REGION Network 11: Trilgoten (4) - Reset Drive
   // Reset van Drive Trilgoten (Drive 2)
   RUNG wire#powerrail
      Contact( "Tag_9" )
      R_Coil( "Drive_2_Auto" )
   END_RUNG
   // the same network as SCL:
   IF "Tag_9" THEN "Drive_2_Auto" := FALSE; END_IF;
END_REGION

REGION Network 12: Aanvoerwals (1) - Set Timing as Drive 1
   RUNG wire#powerrail
      Contact( "PLCMemory".TimingSettingOvername )
      Coil( "Overname_Linked_Drive1" )
   END_RUNG
   // the same network as SCL:
   "Overname_Linked_Drive1" := "PLCMemory".TimingSettingOvername;
END_REGION

REGION Network 13: Aanvoerwals (2) - Run Drive (linked to drive 1)
   RUNG wire#powerrail
      Contact( "Overname_Linked_Drive1" )
      Contact( "Drive_1_Auto" )
      Coil( "Drive_4_Auto" )
   END_RUNG
   // the same network as SCL:
   "Drive_4_Auto" := "Overname_Linked_Drive1" AND "Drive_1_Auto";
END_REGION

REGION Network 14: Aanvoerwals (3) - Set speed Drive 4 (Linked to drive 1)
   RUNG wire#powerrail
      Contact( "PLCMemory".SpeedSettingsTakeover )
      Contact( "Drive 1 Speed 1" )
      Coil( "Drive_4_Speed1_Link" )
   END_RUNG
   // the same network as SCL:
   "Drive_4_Speed1_Link" := "PLCMemory".SpeedSettingsTakeover AND "Drive 1 Speed 1";
END_REGION

REGION Network 15: Aanvoerwals (4) - Set alternative Speed 1
   RUNG wire#powerrail
      I_Contact( "PLCMemory".SpeedSettingsTakeover )
      Contact( "PLCMemory".SpeedSettingOvername )
      I_Contact( "Drive_RefuseLinkingDrive1" )
      Coil( "Drive_4_Speed1_Unlink" )
   END_RUNG
   // the same network as SCL:
   "Drive_4_Speed1_Unlink" := NOT "PLCMemory".SpeedSettingsTakeover AND "PLCMemory".SpeedSettingOvername AND NOT "Drive_RefuseLinkingDrive1";
END_REGION

REGION Network 16: Aanvoerwals (5) - Set alternative Speed 0
   RUNG wire#powerrail
      I_Contact( "PLCMemory".SpeedSettingsTakeover )
      I_Contact( "PLCMemory".SpeedSettingOvername )
      Coil( "Drive_RefuseLinkingDrive1" )
   END_RUNG
   // the same network as SCL:
   "Drive_RefuseLinkingDrive1" := NOT "PLCMemory".SpeedSettingsTakeover AND NOT "PLCMemory".SpeedSettingOvername;
END_REGION

REGION Network 17: Set Position Enable
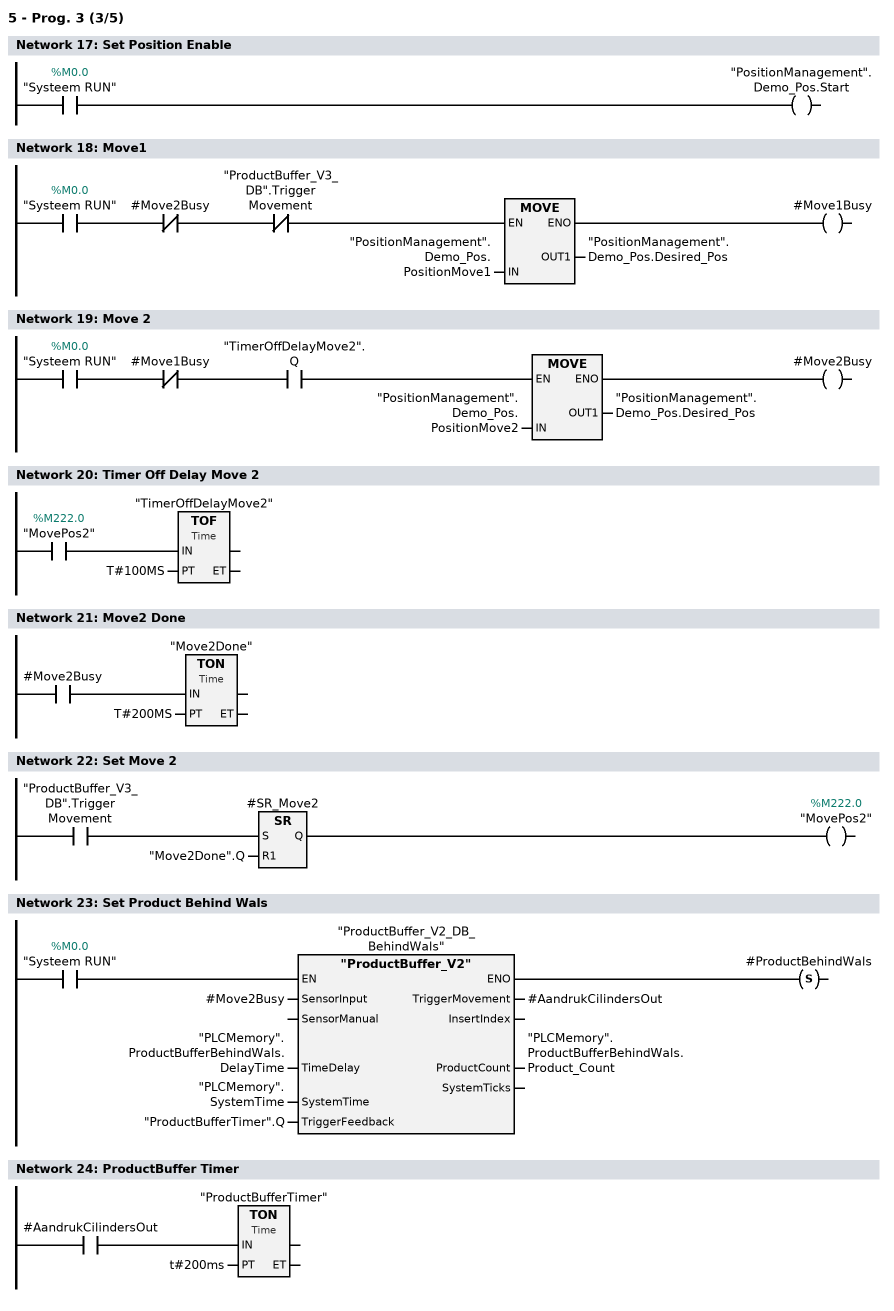
   RUNG wire#powerrail
      Contact( "Systeem RUN" )
      Coil( "PositionManagement".Demo_Pos.Start )
   END_RUNG
   // the same network as SCL:
   "PositionManagement".Demo_Pos.Start := "Systeem RUN";
END_REGION

REGION Network 18: Move1
   RUNG wire#powerrail
      Contact( "Systeem RUN" )
      I_Contact( #Move2Busy )
      I_Contact( "ProductBuffer_V3_DB".TriggerMovement )
      { S7_GenerateENO := "TRUE" } Move(in := "PositionManagement".Demo_Pos.PositionMove1, out1 => "PositionManagement".Demo_Pos.Desired_Pos)
      Coil( #Move1Busy )
   END_RUNG
   // the same network as SCL:
   // ENO of a box is taken as its EN; it also drops when the box reports an error
   #_w1 := "Systeem RUN" AND NOT #Move2Busy AND NOT "ProductBuffer_V3_DB".TriggerMovement;
   IF #_w1 THEN
       "PositionManagement".Demo_Pos.Desired_Pos := "PositionManagement".Demo_Pos.PositionMove1;
   END_IF;
   #Move1Busy := #_w1;
END_REGION

REGION Network 19: Move 2
   RUNG wire#powerrail
      Contact( "Systeem RUN" )
      I_Contact( #Move1Busy )
      Contact( "TimerOffDelayMove2".Q )
      { S7_GenerateENO := "TRUE" } Move(in := "PositionManagement".Demo_Pos.PositionMove2, out1 => "PositionManagement".Demo_Pos.Desired_Pos)
      Coil( #Move2Busy )
   END_RUNG
   // the same network as SCL:
   // ENO of a box is taken as its EN; it also drops when the box reports an error
   #_w1 := "Systeem RUN" AND NOT #Move1Busy AND "TimerOffDelayMove2".Q;
   IF #_w1 THEN
       "PositionManagement".Demo_Pos.Desired_Pos := "PositionManagement".Demo_Pos.PositionMove2;
   END_IF;
   #Move2Busy := #_w1;
END_REGION

REGION Network 20: Timer Off Delay Move 2
   RUNG wire#powerrail
      Contact( "MovePos2" )
      { S7_Templates := "time_type := Time" } "TimerOffDelayMove2".TOF(pt := T#100MS, et =>)
   END_RUNG
   // the same network as SCL:
   "TimerOffDelayMove2".TOF(IN := "MovePos2", PT := T#100MS);
END_REGION

REGION Network 21: Move2 Done
   RUNG wire#powerrail
      Contact( #Move2Busy )
      { S7_Templates := "time_type := Time" } "Move2Done".TON(pt := T#200MS, et =>)
   END_RUNG
   // the same network as SCL:
   "Move2Done".TON(IN := #Move2Busy, PT := T#200MS);
END_REGION

REGION Network 22: Set Move 2
   RUNG wire#powerrail
      Contact( "ProductBuffer_V3_DB".TriggerMovement )
      S_SR(operand := #SR_Move2, r1 := "Move2Done".Q)
      Coil( "MovePos2" )
   END_RUNG
   // the same network as SCL:
   IF "ProductBuffer_V3_DB".TriggerMovement THEN
       #SR_Move2 := TRUE;   // SR flip-flop
   END_IF;
   IF "Move2Done".Q THEN #SR_Move2 := FALSE; END_IF;
   "MovePos2" := #SR_Move2;
END_REGION

REGION Network 23: Set Product Behind Wals
   RUNG wire#powerrail
      Contact( "Systeem RUN" )
      "ProductBuffer_V2_DB_BehindWals"(SensorInput := #Move2Busy, SensorManual :=, TimeDelay := "PLCMemory".ProductBufferBehindWals.DelayTime, SystemTime := "PLCMemory".SystemTime, TriggerFeedback := "ProductBufferTimer".Q, TriggerMovement => #AandrukCilindersOut, InsertIndex =>, ProductCount => "PLCMemory".ProductBufferBehindWals.Product_Count, SystemTicks =>)
      S_Coil( #ProductBehindWals )
   END_RUNG
   // the same network as SCL:
   "ProductBuffer_V2_DB_BehindWals"(EN := "Systeem RUN",   // "ProductBuffer_V2"
                           SensorInput := #Move2Busy,
                           TimeDelay := "PLCMemory".ProductBufferBehindWals.DelayTime,
                           SystemTime := "PLCMemory".SystemTime,
                           TriggerFeedback := "ProductBufferTimer".Q,
                           TriggerMovement => #AandrukCilindersOut,
                           ProductCount => "PLCMemory".ProductBufferBehindWals.Product_Count,
                           ENO => #_w1);
   IF #_w1 THEN #ProductBehindWals := TRUE; END_IF;
END_REGION

REGION Network 24: ProductBuffer Timer
   RUNG wire#powerrail
      Contact( #AandrukCilindersOut )
      { S7_Templates := "time_type := Time" } "ProductBufferTimer".TON(pt := t#200ms, et =>)
   END_RUNG
   // the same network as SCL:
   "ProductBufferTimer".TON(IN := #AandrukCilindersOut, PT := t#200ms);
END_REGION

REGION Network 25: Aandrukken (3) - Outputs
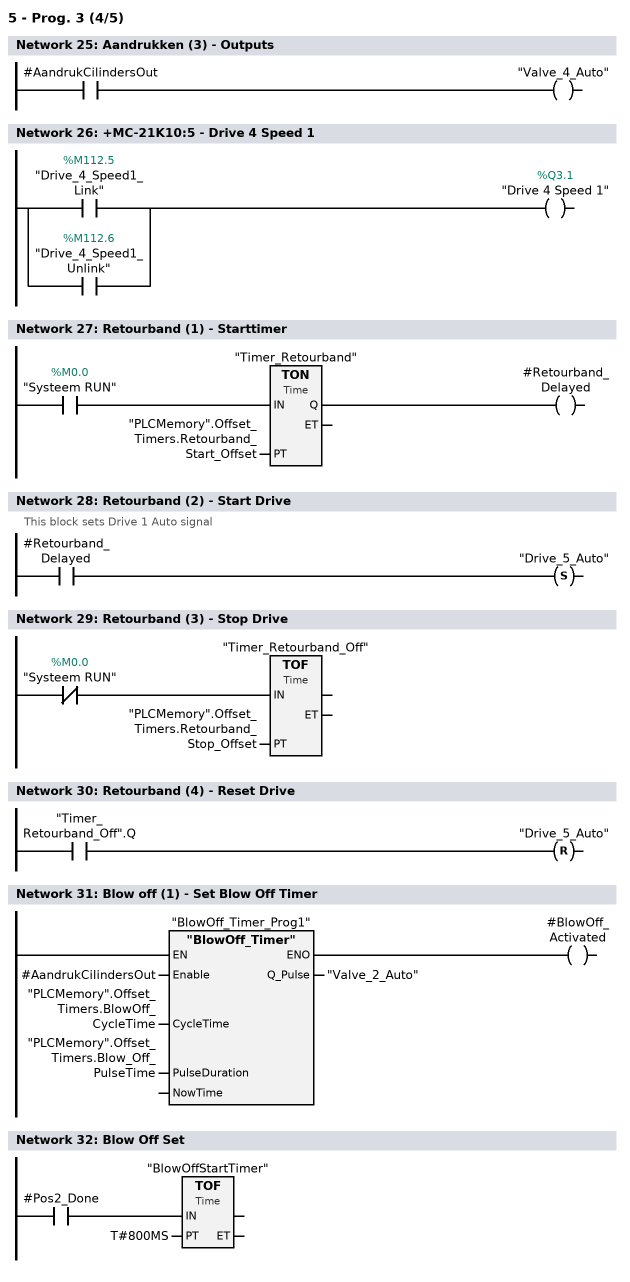
   RUNG wire#powerrail
      Contact( #AandrukCilindersOut )
      Coil( "Valve_4_Auto" )
   END_RUNG
   // the same network as SCL:
   "Valve_4_Auto" := #AandrukCilindersOut;
END_REGION

REGION Network 26: +MC-21K10:5 - Drive 4 Speed 1
   RUNG wire#powerrail
      Contact( "Drive_4_Speed1_Link" )
      wire#w1
      Coil( "Drive 4 Speed 1" )
   END_RUNG
   RUNG wire#powerrail
      Contact( "Drive_4_Speed1_Unlink" )
   END_RUNG wire#w1
   // the same network as SCL:
   "Drive 4 Speed 1" := "Drive_4_Speed1_Link" OR "Drive_4_Speed1_Unlink";
END_REGION

REGION Network 27: Retourband (1) - Starttimer
   RUNG wire#powerrail
      Contact( "Systeem RUN" )
      { S7_Templates := "time_type := Time" } "Timer_Retourband".TON(pt := "PLCMemory".Offset_Timers.Retourband_Start_Offset, et =>)
      Coil( #Retourband_Delayed )
   END_RUNG
   // the same network as SCL:
   "Timer_Retourband".TON(IN := "Systeem RUN", PT := "PLCMemory".Offset_Timers.Retourband_Start_Offset);
   #Retourband_Delayed := "Timer_Retourband".Q;
END_REGION

REGION Network 28: Retourband (2) - Start Drive
   // This block sets Drive 1 Auto signal
   RUNG wire#powerrail
      Contact( #Retourband_Delayed )
      S_Coil( "Drive_5_Auto" )
   END_RUNG
   // the same network as SCL:
   IF #Retourband_Delayed THEN "Drive_5_Auto" := TRUE; END_IF;
END_REGION

REGION Network 29: Retourband (3) - Stop Drive
   RUNG wire#powerrail
      I_Contact( "Systeem RUN" )
      { S7_Templates := "time_type := Time" } "Timer_Retourband_Off".TOF(pt := "PLCMemory".Offset_Timers.Retourband_Stop_Offset, et =>)
   END_RUNG
   // the same network as SCL:
   "Timer_Retourband_Off".TOF(IN := NOT "Systeem RUN", PT := "PLCMemory".Offset_Timers.Retourband_Stop_Offset);
END_REGION

REGION Network 30: Retourband (4) - Reset Drive
   RUNG wire#powerrail
      Contact( "Timer_Retourband_Off".Q )
      R_Coil( "Drive_5_Auto" )
   END_RUNG
   // the same network as SCL:
   IF "Timer_Retourband_Off".Q THEN "Drive_5_Auto" := FALSE; END_IF;
END_REGION

REGION Network 31: Blow off (1) - Set Blow Off Timer
   RUNG wire#powerrail
      "BlowOff_Timer_Prog1"(Enable := #AandrukCilindersOut, CycleTime := "PLCMemory".Offset_Timers.BlowOff_CycleTime, PulseDuration := "PLCMemory".Offset_Timers.Blow_Off_PulseTime, NowTime :=, Q_Pulse => "Valve_2_Auto")
      Coil( #BlowOff_Activated )
   END_RUNG
   // the same network as SCL:
   "BlowOff_Timer_Prog1"(Enable := #AandrukCilindersOut,   // "BlowOff_Timer"
                         CycleTime := "PLCMemory".Offset_Timers.BlowOff_CycleTime,
                         PulseDuration := "PLCMemory".Offset_Timers.Blow_Off_PulseTime,
                         Q_Pulse => "Valve_2_Auto",
                         ENO => #_w1);
   #BlowOff_Activated := #_w1;
END_REGION

REGION Network 32: Blow Off Set
   RUNG wire#powerrail
      Contact( #Pos2_Done )
      { S7_Templates := "time_type := Time" } "BlowOffStartTimer".TOF(pt := T#800MS, et =>)
   END_RUNG
   // the same network as SCL:
   "BlowOffStartTimer".TOF(IN := #Pos2_Done, PT := T#800MS);
END_REGION

REGION Network 33: BlowOffReset
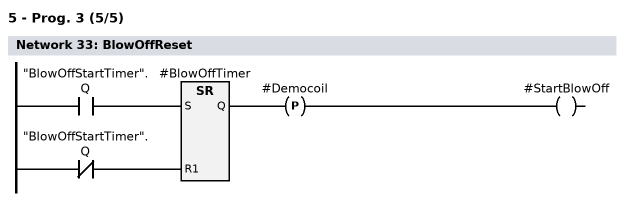
   RUNG wire#powerrail
      Contact( "BlowOffStartTimer".Q )
      S_SR(operand := #BlowOffTimer, r1 := wire#w1)
      P_Trig( #Democoil )
      Coil( #StartBlowOff )
   END_RUNG
   RUNG wire#powerrail
      I_Contact( "BlowOffStartTimer".Q )
   END_RUNG wire#w1
   // the same network as SCL:
   IF "BlowOffStartTimer".Q THEN
       #BlowOffTimer := TRUE;   // SR flip-flop
   END_IF;
   IF NOT "BlowOffStartTimer".Q THEN #BlowOffTimer := FALSE; END_IF;
   #_w1 := #BlowOffTimer AND NOT #Democoil;   // rising edge
   #Democoil := #BlowOffTimer;
   #StartBlowOff := #_w1;
END_REGION
END_FUNCTION

FUNCTION "1 - Outputs" : Void   // FC5, LAD
VERSION : 0.1
// This Function program is for operating the machine automatic and manual.
// stored: AutoNumber true, IsIECCheckEnabled false, UDAEnableTagReadback false
   VAR_TEMP
      Valve_2_Pulse : Bool;
      BlowOff_Activated : Bool;
      BlowOffManual : Bool;
      Pulse1 : Bool;
      Drive_1_ReferenceRun : Bool;
   END_VAR
   VAR_TEMP   // added for the SCL form of the ladder/FBD networks
      _w1 : Bool;
   END_VAR
BEGIN

REGION Network 1: Drive 1 - Control
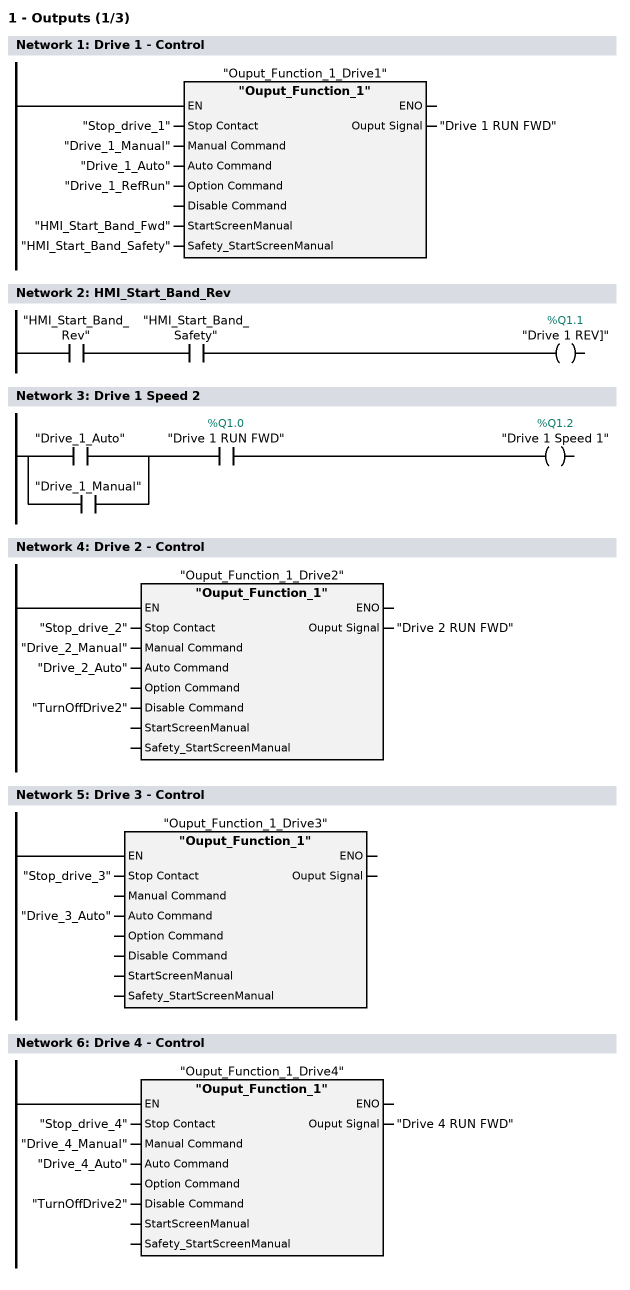
   RUNG wire#powerrail
      "Ouput_Function_1_Drive1"("Stop Contact" := "Stop_drive_1", "Manual Command" := "Drive_1_Manual", "Auto Command" := "Drive_1_Auto", "Option Command" := "Drive_1_RefRun", "Disable Command" :=, StartScreenManual := "HMI_Start_Band_Fwd", Safety_StartScreenManual := "HMI_Start_Band_Safety", "Ouput Signal" => "Drive 1 RUN FWD")
   END_RUNG
   // the same network as SCL:
   "Ouput_Function_1_Drive1"("Stop Contact" := "Stop_drive_1",   // "Ouput_Function_1"
                           "Manual Command" := "Drive_1_Manual",
                           "Auto Command" := "Drive_1_Auto",
                           "Option Command" := "Drive_1_RefRun",
                           StartScreenManual := "HMI_Start_Band_Fwd",
                           Safety_StartScreenManual := "HMI_Start_Band_Safety",
                           "Ouput Signal" => "Drive 1 RUN FWD");
END_REGION

REGION Network 2: HMI_Start_Band_Rev
   RUNG wire#powerrail
      Contact( "HMI_Start_Band_Rev" )
      Contact( "HMI_Start_Band_Safety" )
      Coil( "Drive 1 REV]" )
   END_RUNG
   // the same network as SCL:
   "Drive 1 REV]" := "HMI_Start_Band_Rev" AND "HMI_Start_Band_Safety";
END_REGION

REGION Network 3: Drive 1 Speed 2
   RUNG wire#powerrail
      Contact( "Drive_1_Auto" )
      wire#w1
      Contact( "Drive 1 RUN FWD" )
      Coil( "Drive 1 Speed 1" )
   END_RUNG
   RUNG wire#powerrail
      Contact( "Drive_1_Manual" )
   END_RUNG wire#w1
   // the same network as SCL:
   "Drive 1 Speed 1" := ("Drive_1_Auto" OR "Drive_1_Manual") AND "Drive 1 RUN FWD";
END_REGION

REGION Network 4: Drive 2 - Control
   RUNG wire#powerrail
      "Ouput_Function_1_Drive2"("Stop Contact" := "Stop_drive_2", "Manual Command" := "Drive_2_Manual", "Auto Command" := "Drive_2_Auto", "Option Command" :=, "Disable Command" := "TurnOffDrive2", StartScreenManual :=, Safety_StartScreenManual :=, "Ouput Signal" => "Drive 2 RUN FWD")
   END_RUNG
   // the same network as SCL:
   "Ouput_Function_1_Drive2"("Stop Contact" := "Stop_drive_2",   // "Ouput_Function_1"
                           "Manual Command" := "Drive_2_Manual",
                           "Auto Command" := "Drive_2_Auto",
                           "Disable Command" := "TurnOffDrive2",
                           "Ouput Signal" => "Drive 2 RUN FWD");
END_REGION

REGION Network 5: Drive 3 - Control
   RUNG wire#powerrail
      "Ouput_Function_1_Drive3"("Stop Contact" := "Stop_drive_3", "Manual Command" :=, "Auto Command" := "Drive_3_Auto", "Option Command" :=, "Disable Command" :=, StartScreenManual :=, Safety_StartScreenManual :=, "Ouput Signal" =>)
   END_RUNG
   // the same network as SCL:
   "Ouput_Function_1_Drive3"("Stop Contact" := "Stop_drive_3", "Auto Command" := "Drive_3_Auto");   // "Ouput_Function_1"
END_REGION

REGION Network 6: Drive 4 - Control
   RUNG wire#powerrail
      "Ouput_Function_1_Drive4"("Stop Contact" := "Stop_drive_4", "Manual Command" := "Drive_4_Manual", "Auto Command" := "Drive_4_Auto", "Option Command" :=, "Disable Command" := "TurnOffDrive2", StartScreenManual :=, Safety_StartScreenManual :=, "Ouput Signal" => "Drive 4 RUN FWD")
   END_RUNG
   // the same network as SCL:
   "Ouput_Function_1_Drive4"("Stop Contact" := "Stop_drive_4",   // "Ouput_Function_1"
                           "Manual Command" := "Drive_4_Manual",
                           "Auto Command" := "Drive_4_Auto",
                           "Disable Command" := "TurnOffDrive2",
                           "Ouput Signal" => "Drive 4 RUN FWD");
END_REGION

REGION Network 7: Drive 5 - Control
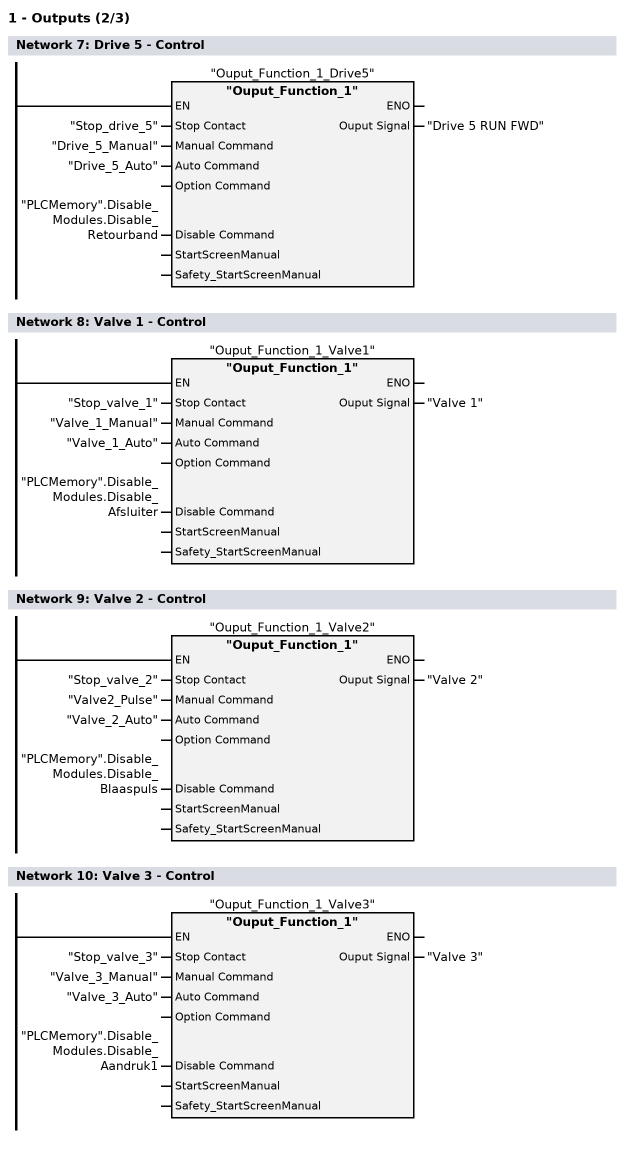
   RUNG wire#powerrail
      "Ouput_Function_1_Drive5"("Stop Contact" := "Stop_drive_5", "Manual Command" := "Drive_5_Manual", "Auto Command" := "Drive_5_Auto", "Option Command" :=, "Disable Command" := "PLCMemory".Disable_Modules.Disable_Retourband, StartScreenManual :=, Safety_StartScreenManual :=, "Ouput Signal" => "Drive 5 RUN FWD")
   END_RUNG
   // the same network as SCL:
   "Ouput_Function_1_Drive5"("Stop Contact" := "Stop_drive_5",   // "Ouput_Function_1"
                           "Manual Command" := "Drive_5_Manual",
                           "Auto Command" := "Drive_5_Auto",
                           "Disable Command" := "PLCMemory".Disable_Modules.Disable_Retourband,
                           "Ouput Signal" => "Drive 5 RUN FWD");
END_REGION

REGION Network 8: Valve 1 - Control
   RUNG wire#powerrail
      "Ouput_Function_1_Valve1"("Stop Contact" := "Stop_valve_1", "Manual Command" := "Valve_1_Manual", "Auto Command" := "Valve_1_Auto", "Option Command" :=, "Disable Command" := "PLCMemory".Disable_Modules.Disable_Afsluiter, StartScreenManual :=, Safety_StartScreenManual :=, "Ouput Signal" => "Valve 1")
   END_RUNG
   // the same network as SCL:
   "Ouput_Function_1_Valve1"("Stop Contact" := "Stop_valve_1",   // "Ouput_Function_1"
                           "Manual Command" := "Valve_1_Manual",
                           "Auto Command" := "Valve_1_Auto",
                           "Disable Command" := "PLCMemory".Disable_Modules.Disable_Afsluiter,
                           "Ouput Signal" => "Valve 1");
END_REGION

REGION Network 9: Valve 2 - Control
   RUNG wire#powerrail
      "Ouput_Function_1_Valve2"("Stop Contact" := "Stop_valve_2", "Manual Command" := "Valve2_Pulse", "Auto Command" := "Valve_2_Auto", "Option Command" :=, "Disable Command" := "PLCMemory".Disable_Modules.Disable_Blaaspuls, StartScreenManual :=, Safety_StartScreenManual :=, "Ouput Signal" => "Valve 2")
   END_RUNG
   // the same network as SCL:
   "Ouput_Function_1_Valve2"("Stop Contact" := "Stop_valve_2",   // "Ouput_Function_1"
                           "Manual Command" := "Valve2_Pulse",
                           "Auto Command" := "Valve_2_Auto",
                           "Disable Command" := "PLCMemory".Disable_Modules.Disable_Blaaspuls,
                           "Ouput Signal" => "Valve 2");
END_REGION

REGION Network 10: Valve 3 - Control
   RUNG wire#powerrail
      "Ouput_Function_1_Valve3"("Stop Contact" := "Stop_valve_3", "Manual Command" := "Valve_3_Manual", "Auto Command" := "Valve_3_Auto", "Option Command" :=, "Disable Command" := "PLCMemory".Disable_Modules.Disable_Aandruk1, StartScreenManual :=, Safety_StartScreenManual :=, "Ouput Signal" => "Valve 3")
   END_RUNG
   // the same network as SCL:
   "Ouput_Function_1_Valve3"("Stop Contact" := "Stop_valve_3",   // "Ouput_Function_1"
                           "Manual Command" := "Valve_3_Manual",
                           "Auto Command" := "Valve_3_Auto",
                           "Disable Command" := "PLCMemory".Disable_Modules.Disable_Aandruk1,
                           "Ouput Signal" => "Valve 3");
END_REGION

REGION Network 11: Valve 4 - Control
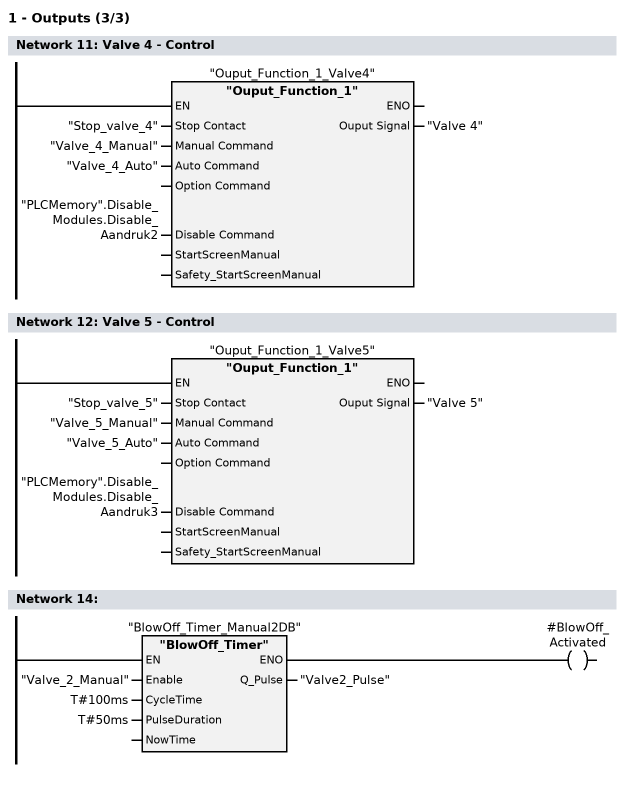
   RUNG wire#powerrail
      "Ouput_Function_1_Valve4"("Stop Contact" := "Stop_valve_4", "Manual Command" := "Valve_4_Manual", "Auto Command" := "Valve_4_Auto", "Option Command" :=, "Disable Command" := "PLCMemory".Disable_Modules.Disable_Aandruk2, StartScreenManual :=, Safety_StartScreenManual :=, "Ouput Signal" => "Valve 4")
   END_RUNG
   // the same network as SCL:
   "Ouput_Function_1_Valve4"("Stop Contact" := "Stop_valve_4",   // "Ouput_Function_1"
                           "Manual Command" := "Valve_4_Manual",
                           "Auto Command" := "Valve_4_Auto",
                           "Disable Command" := "PLCMemory".Disable_Modules.Disable_Aandruk2,
                           "Ouput Signal" => "Valve 4");
END_REGION

REGION Network 12: Valve 5 - Control
   RUNG wire#powerrail
      "Ouput_Function_1_Valve5"("Stop Contact" := "Stop_valve_5", "Manual Command" := "Valve_5_Manual", "Auto Command" := "Valve_5_Auto", "Option Command" :=, "Disable Command" := "PLCMemory".Disable_Modules.Disable_Aandruk3, StartScreenManual :=, Safety_StartScreenManual :=, "Ouput Signal" => "Valve 5")
   END_RUNG
   // the same network as SCL:
   "Ouput_Function_1_Valve5"("Stop Contact" := "Stop_valve_5",   // "Ouput_Function_1"
                           "Manual Command" := "Valve_5_Manual",
                           "Auto Command" := "Valve_5_Auto",
                           "Disable Command" := "PLCMemory".Disable_Modules.Disable_Aandruk3,
                           "Ouput Signal" => "Valve 5");
END_REGION

REGION Network 13: Blow Off Manual
END_REGION

REGION Network 14
   RUNG wire#powerrail
      "BlowOff_Timer_Manual2DB"(Enable := "Valve_2_Manual", CycleTime := T#100ms, PulseDuration := T#50ms, NowTime :=, Q_Pulse => "Valve2_Pulse")
      Coil( #BlowOff_Activated )
   END_RUNG
   // the same network as SCL:
   "BlowOff_Timer_Manual2DB"(Enable := "Valve_2_Manual",   // "BlowOff_Timer"
                           CycleTime := T#100ms,
                           PulseDuration := T#50ms,
                           Q_Pulse => "Valve2_Pulse",
                           ENO => #_w1);
   #BlowOff_Activated := #_w1;
END_REGION
END_FUNCTION

FUNCTION_BLOCK "Ouput_Function_1"   // FB8, FBD
TITLE = Ouput Controller Function Block
VERSION : 0.1
// stored: AutoNumber true, IsIECCheckEnabled false, UDAEnableTagReadback false
   VAR_INPUT
      "Stop Contact" : Bool;
      "Manual Command" : Bool;
      "Auto Command" : Bool;
      "Option Command" : Bool;
      "Disable Command" : Bool;
      StartScreenManual : Bool;
      Safety_StartScreenManual : Bool;
   END_VAR
   VAR_OUTPUT
      "Ouput Signal" : Bool;
   END_VAR
BEGIN

REGION Network 1: Ouput Controller
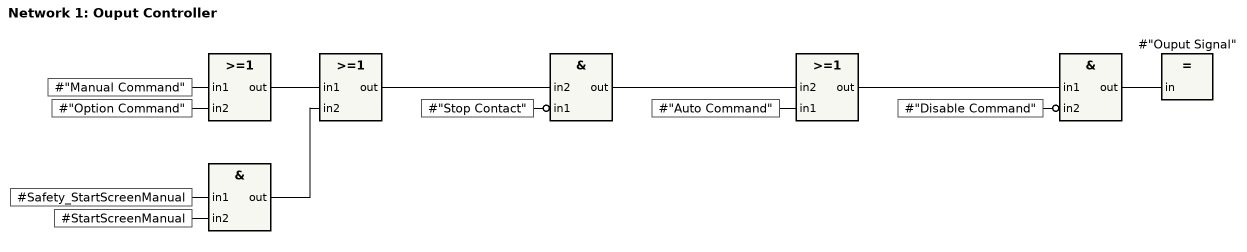
   #"Ouput Signal" := (((#"Manual Command" OR #"Option Command" OR (#Safety_StartScreenManual AND #StartScreenManual)) AND NOT #"Stop Contact") OR #"Auto Command") AND NOT #"Disable Command";
END_REGION
END_FUNCTION_BLOCK

FUNCTION "6 - Storingsmelding" : Void   // FC8, LAD
TITLE = Warnings
VERSION : 0.1
// This program block is for audible & visual warnings.
// stored: AutoNumber true, IsIECCheckEnabled false, UDAEnableTagReadback false
   VAR_TEMP
      "Wals Sensor Controlled" : Bool;
      "Infeed Sensor Controlled" : Bool;
      EnoughProductsOnInfeed : Bool;
      NotEnoughProductsOnInfeed : Bool;
      Warning_NotEnoughProducts : Bool;
      TurnOffDrives : Bool;
   END_VAR
   VAR CONSTANT
      "Sensor 2 (option)" : Bool := TRUE;
   END_VAR
   VAR_TEMP   // added for the SCL form of the ladder/FBD networks
      _w1 : Bool;
   END_VAR
BEGIN

REGION Network 1: +MC-21K6:5 - Bel Storing
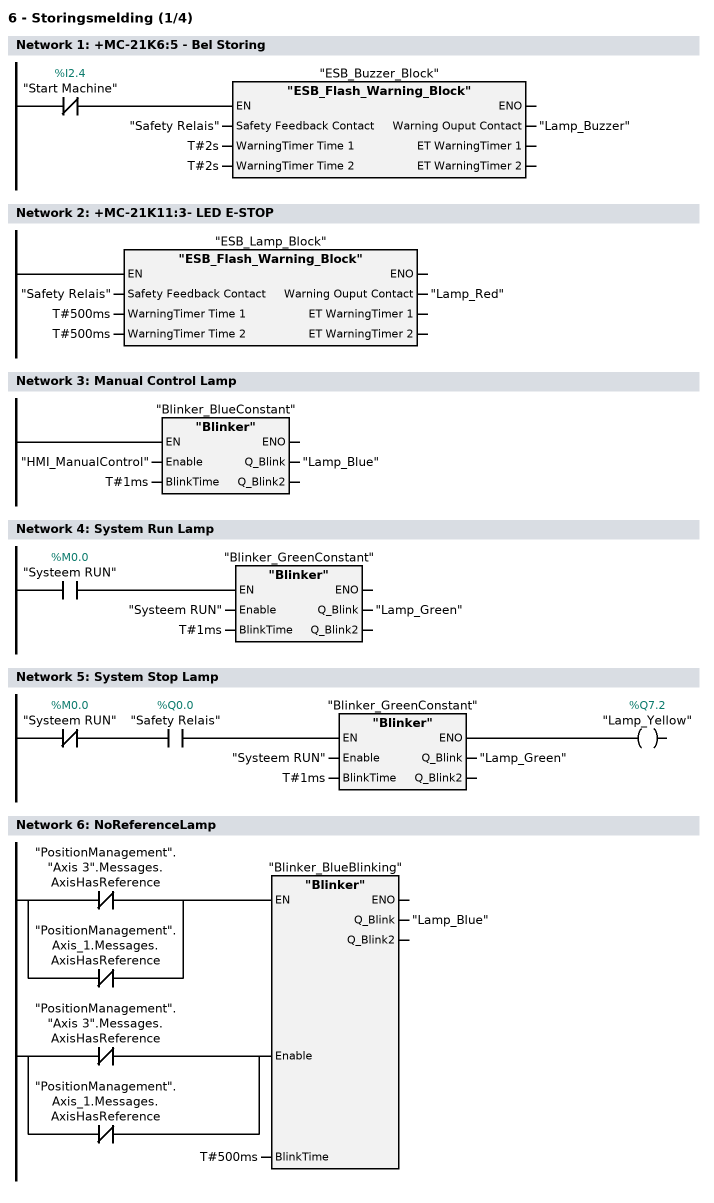
   RUNG wire#powerrail
      I_Contact( "Start Machine" )
      "ESB_Buzzer_Block"("Safety Feedback Contact" := "Safety Relais", "WarningTimer Time 1" := T#2s, "WarningTimer Time 2" := T#2s, "Warning Ouput Contact" => "Lamp_Buzzer", "ET WarningTimer 1" =>, "ET WarningTimer 2" =>)
   END_RUNG
   // the same network as SCL:
   IF NOT "Start Machine" THEN
       "ESB_Buzzer_Block"("Safety Feedback Contact" := "Safety Relais",   // "ESB_Flash_Warning_Block"
                          "WarningTimer Time 1" := T#2s,
                          "WarningTimer Time 2" := T#2s,
                          "Warning Ouput Contact" => "Lamp_Buzzer");
   END_IF;
END_REGION

REGION Network 2: +MC-21K11:3- LED E-STOP
   RUNG wire#powerrail
      "ESB_Lamp_Block"("Safety Feedback Contact" := "Safety Relais", "WarningTimer Time 1" := T#500ms, "WarningTimer Time 2" := T#500ms, "Warning Ouput Contact" => "Lamp_Red", "ET WarningTimer 1" =>, "ET WarningTimer 2" =>)
   END_RUNG
   // the same network as SCL:
   "ESB_Lamp_Block"("Safety Feedback Contact" := "Safety Relais",   // "ESB_Flash_Warning_Block"
                    "WarningTimer Time 1" := T#500ms,
                    "WarningTimer Time 2" := T#500ms,
                    "Warning Ouput Contact" => "Lamp_Red");
END_REGION

REGION Network 3: Manual Control Lamp
   RUNG wire#powerrail
      "Blinker_BlueConstant"(Enable := "HMI_ManualControl", BlinkTime := T#1ms, Q_Blink => "Lamp_Blue", Q_Blink2 =>)
   END_RUNG
   // the same network as SCL:
   "Blinker_BlueConstant"(Enable := "HMI_ManualControl", BlinkTime := T#1ms, Q_Blink => "Lamp_Blue");   // "Blinker"
END_REGION

REGION Network 4: System Run Lamp
   RUNG wire#powerrail
      Contact( "Systeem RUN" )
      "Blinker_GreenConstant"(Enable := "Systeem RUN", BlinkTime := T#1ms, Q_Blink => "Lamp_Green", Q_Blink2 =>)
   END_RUNG
   // the same network as SCL:
   IF "Systeem RUN" THEN
       "Blinker_GreenConstant"(Enable := "Systeem RUN", BlinkTime := T#1ms, Q_Blink => "Lamp_Green");   // "Blinker"
   END_IF;
END_REGION

REGION Network 5: System Stop Lamp
   RUNG wire#powerrail
      I_Contact( "Systeem RUN" )
      Contact( "Safety Relais" )
      "Blinker_GreenConstant"(Enable := "Systeem RUN", BlinkTime := T#1ms, Q_Blink => "Lamp_Green", Q_Blink2 =>)
      Coil( "Lamp_Yellow" )
   END_RUNG
   // the same network as SCL:
   "Blinker_GreenConstant"(EN := NOT "Systeem RUN" AND "Safety Relais",   // "Blinker"
                           Enable := "Systeem RUN",
                           BlinkTime := T#1ms,
                           Q_Blink => "Lamp_Green",
                           ENO => #_w1);
   "Lamp_Yellow" := #_w1;
END_REGION

REGION Network 6: NoReferenceLamp
   RUNG wire#powerrail
      I_Contact( "PositionManagement"."Axis 3".Messages.AxisHasReference )
      wire#w1
      "Blinker_BlueBlinking"(Enable := wire#w2, BlinkTime := T#500ms, Q_Blink => "Lamp_Blue", Q_Blink2 =>)
   END_RUNG
   RUNG wire#powerrail
      I_Contact( "PositionManagement".Axis_1.Messages.AxisHasReference )
   END_RUNG wire#w1
   RUNG wire#powerrail
      I_Contact( "PositionManagement"."Axis 3".Messages.AxisHasReference )
   END_RUNG wire#w2
   RUNG wire#powerrail
      I_Contact( "PositionManagement".Axis_1.Messages.AxisHasReference )
   END_RUNG wire#w2
   // the same network as SCL:
   IF NOT "PositionManagement"."Axis 3".Messages.AxisHasReference OR NOT "PositionManagement".Axis_1.Messages.AxisHasReference THEN
       "Blinker_BlueBlinking"(Enable := NOT "PositionManagement"."Axis 3".Messages.AxisHasReference OR NOT "PositionManagement".Axis_1.Messages.AxisHasReference,   // "Blinker"
                              BlinkTime := T#500ms,
                              Q_Blink => "Lamp_Blue");
   END_IF;
END_REGION

REGION Network 7: Fill Trechter Delay Function
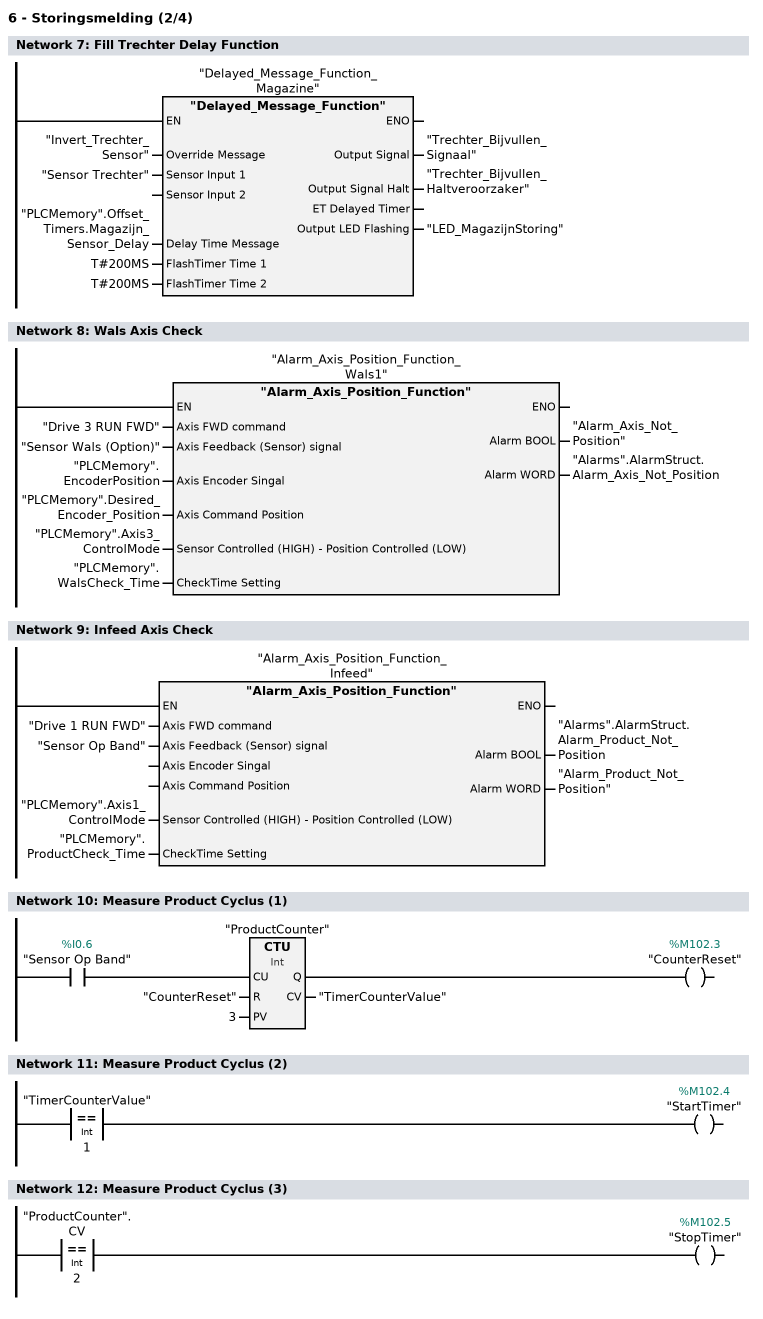
   RUNG wire#powerrail
      "Delayed_Message_Function_Magazine"("Override Message" := "Invert_Trechter_Sensor", "Sensor Input 1" := "Sensor Trechter", "Sensor Input 2" :=, "Delay Time Message" := "PLCMemory".Offset_Timers.Magazijn_Sensor_Delay, "FlashTimer Time 1" := T#200MS, "FlashTimer Time 2" := T#200MS, "Output Signal" => "Trechter_Bijvullen_Signaal", "Output Signal Halt" => "Trechter_Bijvullen_Haltveroorzaker", "ET Delayed Timer" =>, "Output LED Flashing" => "LED_MagazijnStoring")
   END_RUNG
   // the same network as SCL:
   "Delayed_Message_Function_Magazine"("Override Message" := "Invert_Trechter_Sensor",   // "Delayed_Message_Function"
                           "Sensor Input 1" := "Sensor Trechter",
                           "Delay Time Message" := "PLCMemory".Offset_Timers.Magazijn_Sensor_Delay,
                           "FlashTimer Time 1" := T#200MS,
                           "FlashTimer Time 2" := T#200MS,
                           "Output Signal" => "Trechter_Bijvullen_Signaal",
                           "Output Signal Halt" => "Trechter_Bijvullen_Haltveroorzaker",
                           "Output LED Flashing" => "LED_MagazijnStoring");
END_REGION

REGION Network 8: Wals Axis Check
   RUNG wire#powerrail
      "Alarm_Axis_Position_Function_Wals1"("Axis FWD command" := "Drive 3 RUN FWD", "Axis Feedback (Sensor) signal" := "Sensor Wals (Option)", "Axis Encoder Singal" := "PLCMemory".EncoderPosition, "Axis Command Position" := "PLCMemory".Desired_Encoder_Position, "Sensor Controlled (HIGH) - Position Controlled (LOW)" := "PLCMemory".Axis3_ControlMode, "CheckTime Setting" := "PLCMemory".WalsCheck_Time, "Alarm BOOL" => "Alarm_Axis_Not_Position", "Alarm WORD" => "Alarms".AlarmStruct.Alarm_Axis_Not_Position)
   END_RUNG
   // the same network as SCL:
   "Alarm_Axis_Position_Function_Wals1"("Axis FWD command" := "Drive 3 RUN FWD",   // "Alarm_Axis_Position_Function"
                           "Axis Feedback (Sensor) signal" := "Sensor Wals (Option)",
                           "Axis Encoder Singal" := "PLCMemory".EncoderPosition,
                           "Axis Command Position" := "PLCMemory".Desired_Encoder_Position,
                           "Sensor Controlled (HIGH) - Position Controlled (LOW)" := "PLCMemory".Axis3_ControlMode,
                           "CheckTime Setting" := "PLCMemory".WalsCheck_Time,
                           "Alarm BOOL" => "Alarm_Axis_Not_Position",
                           "Alarm WORD" => "Alarms".AlarmStruct.Alarm_Axis_Not_Position);
END_REGION

REGION Network 9: Infeed Axis Check
   RUNG wire#powerrail
      "Alarm_Axis_Position_Function_Infeed"("Axis FWD command" := "Drive 1 RUN FWD", "Axis Feedback (Sensor) signal" := "Sensor Op Band", "Axis Encoder Singal" :=, "Axis Command Position" :=, "Sensor Controlled (HIGH) - Position Controlled (LOW)" := "PLCMemory".Axis1_ControlMode, "CheckTime Setting" := "PLCMemory".ProductCheck_Time, "Alarm BOOL" => "Alarms".AlarmStruct.Alarm_Product_Not_Position, "Alarm WORD" => "Alarm_Product_Not_Position")
   END_RUNG
   // the same network as SCL:
   "Alarm_Axis_Position_Function_Infeed"("Axis FWD command" := "Drive 1 RUN FWD",   // "Alarm_Axis_Position_Function"
                           "Axis Feedback (Sensor) signal" := "Sensor Op Band",
                           "Sensor Controlled (HIGH) - Position Controlled (LOW)" := "PLCMemory".Axis1_ControlMode,
                           "CheckTime Setting" := "PLCMemory".ProductCheck_Time,
                           "Alarm BOOL" => "Alarms".AlarmStruct.Alarm_Product_Not_Position,
                           "Alarm WORD" => "Alarm_Product_Not_Position");
END_REGION

REGION Network 10: Measure Product Cyclus (1)
   RUNG wire#powerrail
      Contact( "Sensor Op Band" )
      { S7_Templates := "value_type := Int" } "ProductCounter".CTU(r := "CounterReset", pv := 3, cv => "TimerCounterValue")
      Coil( "CounterReset" )
   END_RUNG
   // the same network as SCL:
   "ProductCounter".CTU(CU := "Sensor Op Band", R := "CounterReset", PV := 3, CV => "TimerCounterValue");
   "CounterReset" := "ProductCounter".Q;
END_REGION

REGION Network 11: Measure Product Cyclus (2)
   RUNG wire#powerrail
      { S7_Templates := "SrcType := Int" } EQ_Contact(in1 := "TimerCounterValue", in2 := 1)
      Coil( "StartTimer" )
   END_RUNG
   // the same network as SCL:
   "StartTimer" := "TimerCounterValue" = 1;
END_REGION

REGION Network 12: Measure Product Cyclus (3)
   RUNG wire#powerrail
      { S7_Templates := "SrcType := Int" } EQ_Contact(in1 := "ProductCounter".CV, in2 := 2)
      Coil( "StopTimer" )
   END_RUNG
   // the same network as SCL:
   "StopTimer" := "ProductCounter".CV = 2;
END_REGION

REGION Network 13: Measure Product Cyclus (4)
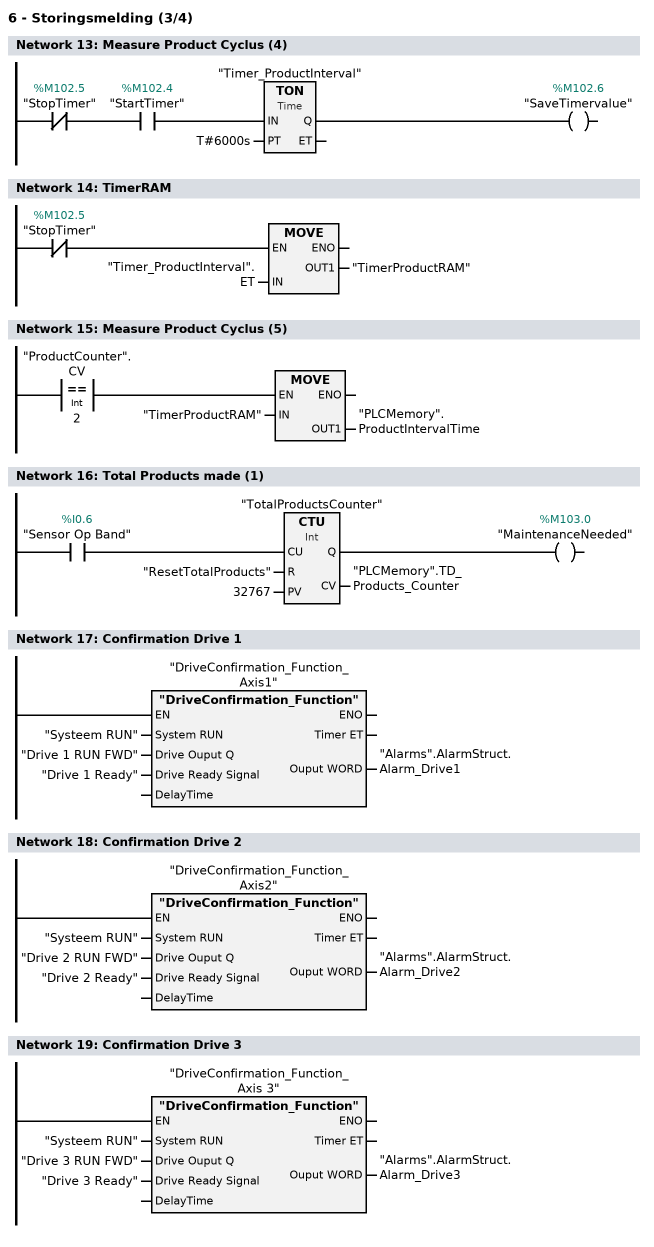
   RUNG wire#powerrail
      I_Contact( "StopTimer" )
      Contact( "StartTimer" )
      { S7_Templates := "time_type := Time" } "Timer_ProductInterval".TON(pt := T#6000s, et =>)
      Coil( "SaveTimervalue" )
   END_RUNG
   // the same network as SCL:
   "Timer_ProductInterval".TON(IN := NOT "StopTimer" AND "StartTimer", PT := T#6000s);
   "SaveTimervalue" := "Timer_ProductInterval".Q;
END_REGION

REGION Network 14: TimerRAM
   RUNG wire#powerrail
      I_Contact( "StopTimer" )
      { S7_GenerateENO := "TRUE" } Move(in := "Timer_ProductInterval".ET, out1 => "TimerProductRAM")
   END_RUNG
   // the same network as SCL:
   IF NOT "StopTimer" THEN "TimerProductRAM" := "Timer_ProductInterval".ET; END_IF;
END_REGION

REGION Network 15: Measure Product Cyclus (5)
   RUNG wire#powerrail
      { S7_Templates := "SrcType := Int" } EQ_Contact(in1 := "ProductCounter".CV, in2 := 2)
      { S7_GenerateENO := "TRUE" } Move(in := "TimerProductRAM", out1 => "PLCMemory".ProductIntervalTime)
   END_RUNG
   // the same network as SCL:
   IF "ProductCounter".CV = 2 THEN "PLCMemory".ProductIntervalTime := "TimerProductRAM"; END_IF;
END_REGION

REGION Network 16: Total Products made (1)
   RUNG wire#powerrail
      Contact( "Sensor Op Band" )
      { S7_Templates := "value_type := Int" } "TotalProductsCounter".CTU(r := "ResetTotalProducts", pv := 32767, cv => "PLCMemory".TD_Products_Counter)
      Coil( "MaintenanceNeeded" )
   END_RUNG
   // the same network as SCL:
   "TotalProductsCounter".CTU(CU := "Sensor Op Band",
                           R := "ResetTotalProducts",
                           PV := 32767,
                           CV => "PLCMemory".TD_Products_Counter);
   "MaintenanceNeeded" := "TotalProductsCounter".Q;
END_REGION

REGION Network 17: Confirmation Drive 1
   RUNG wire#powerrail
      "DriveConfirmation_Function_Axis1"("System RUN" := "Systeem RUN", "Drive Ouput Q" := "Drive 1 RUN FWD", "Drive Ready Signal" := "Drive 1 Ready", DelayTime :=, "Timer ET" =>, "Ouput WORD" => "Alarms".AlarmStruct.Alarm_Drive1)
   END_RUNG
   // the same network as SCL:
   "DriveConfirmation_Function_Axis1"("System RUN" := "Systeem RUN",   // "DriveConfirmation_Function"
                           "Drive Ouput Q" := "Drive 1 RUN FWD",
                           "Drive Ready Signal" := "Drive 1 Ready",
                           "Ouput WORD" => "Alarms".AlarmStruct.Alarm_Drive1);
END_REGION

REGION Network 18: Confirmation Drive 2
   RUNG wire#powerrail
      "DriveConfirmation_Function_Axis2"("System RUN" := "Systeem RUN", "Drive Ouput Q" := "Drive 2 RUN FWD", "Drive Ready Signal" := "Drive 2 Ready", DelayTime :=, "Timer ET" =>, "Ouput WORD" => "Alarms".AlarmStruct.Alarm_Drive2)
   END_RUNG
   // the same network as SCL:
   "DriveConfirmation_Function_Axis2"("System RUN" := "Systeem RUN",   // "DriveConfirmation_Function"
                           "Drive Ouput Q" := "Drive 2 RUN FWD",
                           "Drive Ready Signal" := "Drive 2 Ready",
                           "Ouput WORD" => "Alarms".AlarmStruct.Alarm_Drive2);
END_REGION

REGION Network 19: Confirmation Drive 3
   RUNG wire#powerrail
      "DriveConfirmation_Function_Axis 3"("System RUN" := "Systeem RUN", "Drive Ouput Q" := "Drive 3 RUN FWD", "Drive Ready Signal" := "Drive 3 Ready", DelayTime :=, "Timer ET" =>, "Ouput WORD" => "Alarms".AlarmStruct.Alarm_Drive3)
   END_RUNG
   // the same network as SCL:
   "DriveConfirmation_Function_Axis 3"("System RUN" := "Systeem RUN",   // "DriveConfirmation_Function"
                           "Drive Ouput Q" := "Drive 3 RUN FWD",
                           "Drive Ready Signal" := "Drive 3 Ready",
                           "Ouput WORD" => "Alarms".AlarmStruct.Alarm_Drive3);
END_REGION

REGION Network 20: Confimation Drive 4
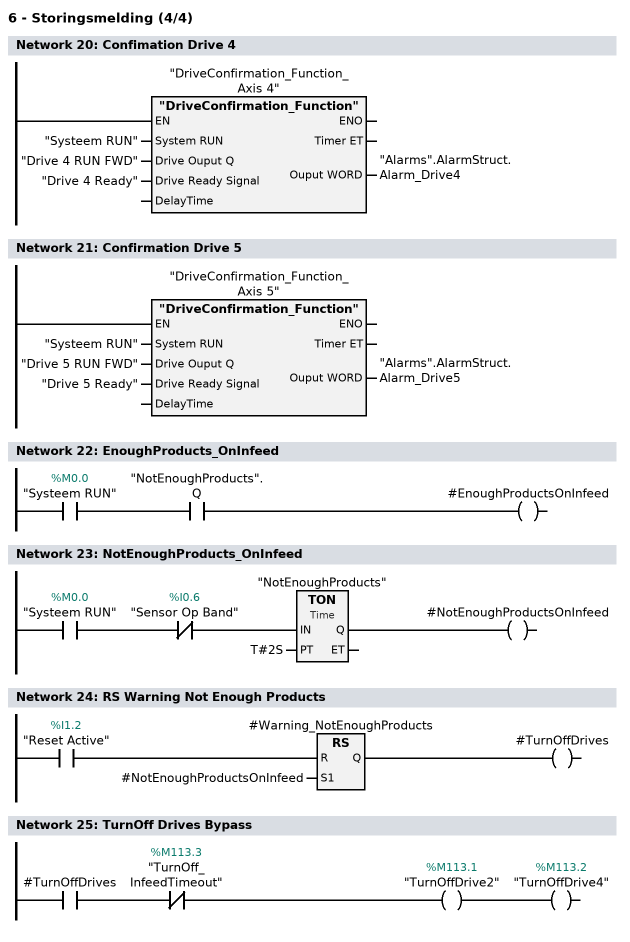
   RUNG wire#powerrail
      "DriveConfirmation_Function_Axis 4"("System RUN" := "Systeem RUN", "Drive Ouput Q" := "Drive 4 RUN FWD", "Drive Ready Signal" := "Drive 4 Ready", DelayTime :=, "Timer ET" =>, "Ouput WORD" => "Alarms".AlarmStruct.Alarm_Drive4)
   END_RUNG
   // the same network as SCL:
   "DriveConfirmation_Function_Axis 4"("System RUN" := "Systeem RUN",   // "DriveConfirmation_Function"
                           "Drive Ouput Q" := "Drive 4 RUN FWD",
                           "Drive Ready Signal" := "Drive 4 Ready",
                           "Ouput WORD" => "Alarms".AlarmStruct.Alarm_Drive4);
END_REGION

REGION Network 21: Confirmation Drive 5
   RUNG wire#powerrail
      "DriveConfirmation_Function_Axis 5"("System RUN" := "Systeem RUN", "Drive Ouput Q" := "Drive 5 RUN FWD", "Drive Ready Signal" := "Drive 5 Ready", DelayTime :=, "Timer ET" =>, "Ouput WORD" => "Alarms".AlarmStruct.Alarm_Drive5)
   END_RUNG
   // the same network as SCL:
   "DriveConfirmation_Function_Axis 5"("System RUN" := "Systeem RUN",   // "DriveConfirmation_Function"
                           "Drive Ouput Q" := "Drive 5 RUN FWD",
                           "Drive Ready Signal" := "Drive 5 Ready",
                           "Ouput WORD" => "Alarms".AlarmStruct.Alarm_Drive5);
END_REGION

REGION Network 22: EnoughProducts_OnInfeed
   RUNG wire#powerrail
      Contact( "Systeem RUN" )
      Contact( "NotEnoughProducts".Q )
      Coil( #EnoughProductsOnInfeed )
   END_RUNG
   // the same network as SCL:
   #EnoughProductsOnInfeed := "Systeem RUN" AND "NotEnoughProducts".Q;
END_REGION

REGION Network 23: NotEnoughProducts_OnInfeed
   RUNG wire#powerrail
      Contact( "Systeem RUN" )
      I_Contact( "Sensor Op Band" )
      { S7_Templates := "time_type := Time" } "NotEnoughProducts".TON(pt := T#2S, et =>)
      Coil( #NotEnoughProductsOnInfeed )
   END_RUNG
   // the same network as SCL:
   "NotEnoughProducts".TON(IN := "Systeem RUN" AND NOT "Sensor Op Band", PT := T#2S);
   #NotEnoughProductsOnInfeed := "NotEnoughProducts".Q;
END_REGION

REGION Network 24: RS Warning Not Enough Products
   RUNG wire#powerrail
      Contact( "Reset Active" )
      S_RS(operand := #Warning_NotEnoughProducts, s1 := #NotEnoughProductsOnInfeed)
      Coil( #TurnOffDrives )
   END_RUNG
   // the same network as SCL:
   IF "Reset Active" THEN
       #Warning_NotEnoughProducts := FALSE;   // RS flip-flop
   END_IF;
   IF #NotEnoughProductsOnInfeed THEN #Warning_NotEnoughProducts := TRUE; END_IF;
   #TurnOffDrives := #Warning_NotEnoughProducts;
END_REGION

REGION Network 25: TurnOff Drives Bypass
   RUNG wire#powerrail
      Contact( #TurnOffDrives )
      I_Contact( "TurnOff_InfeedTimeout" )
      Coil( "TurnOffDrive2" )
      Coil( "TurnOffDrive4" )
   END_RUNG
   // the same network as SCL:
   "TurnOffDrive2" := #TurnOffDrives AND NOT "TurnOff_InfeedTimeout";
   "TurnOffDrive4" := "TurnOffDrive2";
END_REGION
END_FUNCTION

FUNCTION_BLOCK "ESB_Flash_Warning_Block"   // FB1, FBD
VERSION : 0.1
// stored: AutoNumber true, IsIECCheckEnabled false, UDAEnableTagReadback false
   VAR_INPUT
      "Safety Feedback Contact" : Bool;
      "WarningTimer Time 1" : Time := T#150ms;
      "WarningTimer Time 2" : Time := T#150ms;
   END_VAR
   VAR_OUTPUT
      "Warning Ouput Contact" : Bool;
      "ET WarningTimer 1" : Time;
      "ET WarningTimer 2" : Time;
   END_VAR
   VAR_TEMP
      SafetyTakeoverContact : Bool;
   END_VAR
   VAR_TEMP   // added for the SCL form of the ladder/FBD networks
      _w1 : Bool;
   END_VAR
BEGIN

REGION Network 1: Flash Warning
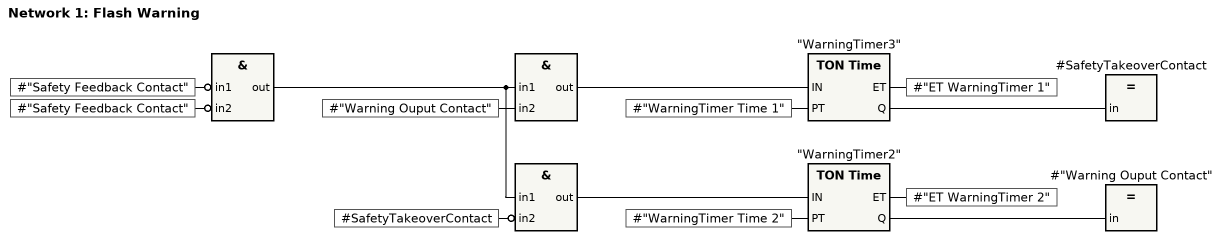
   #_w1 := NOT #"Safety Feedback Contact" AND NOT #"Safety Feedback Contact";
   "WarningTimer3".TON(IN := #_w1 AND #"Warning Ouput Contact",
                       PT := #"WarningTimer Time 1",
                       ET => #"ET WarningTimer 1");
   #SafetyTakeoverContact := "WarningTimer3".Q;
   "WarningTimer2".TON(IN := #_w1 AND NOT #SafetyTakeoverContact,
                       PT := #"WarningTimer Time 2",
                       ET => #"ET WarningTimer 2");
   #"Warning Ouput Contact" := "WarningTimer2".Q;
END_REGION
END_FUNCTION_BLOCK

FUNCTION_BLOCK "Delayed_Message_Function"   // FB2, FBD
TITLE = Delayed Message Function
VERSION : 0.1
// Functionblock For Delaying Message Function for example for filling an magazine or waiting for an signal. It is possible to adjust Time with the Dleay Time Message Input. The FlashTimer Time 1 & 2 ar for adjusting the flashing time of the ouput LED.
// stored: AutoNumber true, IsIECCheckEnabled false, UDAEnableTagReadback false
   VAR_INPUT
      "Override Message" : Bool;
      "Sensor Input 1" : Bool;
      "Sensor Input 2" : Bool := true;
      "Delay Time Message" : Time := T#1S_500MS;
      "FlashTimer Time 1" : Time := T#200ms;
      "FlashTimer Time 2" : Time := T#200ms;
   END_VAR
   VAR_OUTPUT
      "Output Signal" : Bool;
      "Output Signal Halt" : Bool;
      "ET Delayed Timer" : Time;
      "Output LED Flashing" : Bool;
   END_VAR
   VAR_TEMP
      "Internal Delayed Signal" : Bool;
   END_VAR
   VAR_TEMP   // added for the SCL form of the ladder/FBD networks
      _w1 : Bool;
   END_VAR
BEGIN

REGION Network 1: Delayed Signal to Outputs
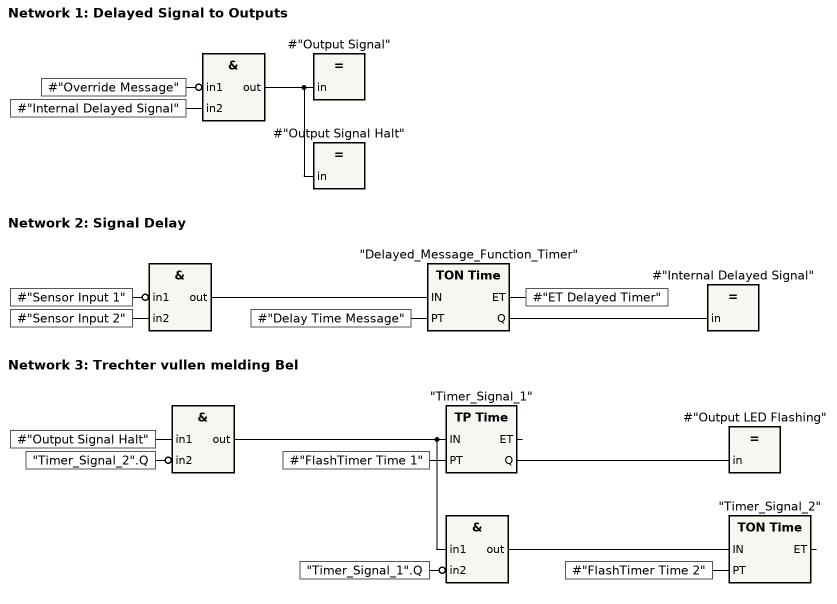
   #"Output Signal" := NOT #"Override Message" AND #"Internal Delayed Signal";
   #"Output Signal Halt" := #"Output Signal";
END_REGION

REGION Network 2: Signal Delay
   "Delayed_Message_Function_Timer".TON(IN := NOT #"Sensor Input 1" AND #"Sensor Input 2",
                           PT := #"Delay Time Message",
                           ET => #"ET Delayed Timer");
   #"Internal Delayed Signal" := "Delayed_Message_Function_Timer".Q;
END_REGION

REGION Network 3: Trechter vullen melding Bel
   #_w1 := #"Output Signal Halt" AND NOT "Timer_Signal_2".Q;
   "Timer_Signal_1".TP(IN := #_w1, PT := #"FlashTimer Time 1");
   #"Output LED Flashing" := "Timer_Signal_1".Q;
   "Timer_Signal_2".TON(IN := #_w1 AND NOT "Timer_Signal_1".Q, PT := #"FlashTimer Time 2");
END_REGION
END_FUNCTION_BLOCK

FUNCTION_BLOCK "Alarm_Axis_Position_Function"   // FB3, FBD
TITLE = Alarm Axis not in Position
VERSION : 0.1
// stored: AutoNumber true, IsIECCheckEnabled false, UDAEnableTagReadback false
   VAR_INPUT
      "Axis FWD command" : Bool;
      "Axis Feedback (Sensor) signal" : Bool;
      "Axis Encoder Singal" : Real;
      "Axis Command Position" : Real;
      "Sensor Controlled (HIGH) - Position Controlled (LOW)" : Bool;
      "CheckTime Setting" : Time := T#5S;
   END_VAR
   VAR_OUTPUT
      "Alarm BOOL" : Bool;
      "Alarm WORD" : Bool;
   END_VAR
   VAR_TEMP
      "Axis Feedback Internal" : Bool;
      "Axis Encoder On Position" : Bool;
      "Axis Sensor On Position" : Bool;
      "Axis Measuring Mode" : Bool;
   END_VAR
BEGIN

REGION Network 1: When axis is spinning start timer
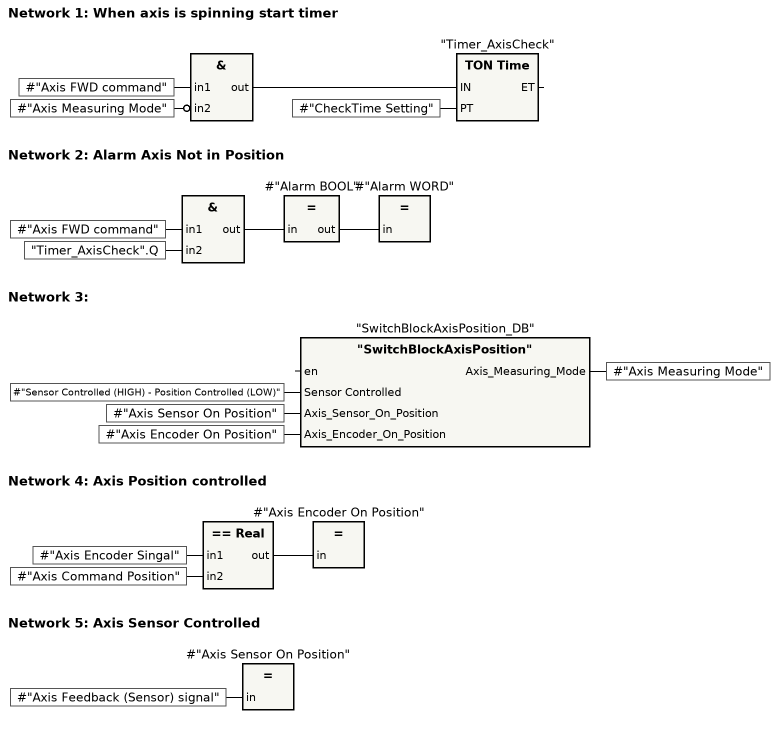
   "Timer_AxisCheck".TON(IN := #"Axis FWD command" AND NOT #"Axis Measuring Mode", PT := #"CheckTime Setting");
END_REGION

REGION Network 2: Alarm Axis Not in Position
   #"Alarm BOOL" := #"Axis FWD command" AND "Timer_AxisCheck".Q;
   #"Alarm WORD" := #"Alarm BOOL";
END_REGION

REGION Network 3
   "SwitchBlockAxisPosition_DB"("Sensor Controlled" := #"Sensor Controlled (HIGH) - Position Controlled (LOW)",   // "SwitchBlockAxisPosition"
                           Axis_Sensor_On_Position := #"Axis Sensor On Position",
                           Axis_Encoder_On_Position := #"Axis Encoder On Position",
                           Axis_Measuring_Mode => #"Axis Measuring Mode");
END_REGION

REGION Network 4: Axis Position controlled
   #"Axis Encoder On Position" := #"Axis Encoder Singal" = #"Axis Command Position";
END_REGION

REGION Network 5: Axis Sensor Controlled
   #"Axis Sensor On Position" := #"Axis Feedback (Sensor) signal";
END_REGION
END_FUNCTION_BLOCK

FUNCTION_BLOCK "SwitchBlockAxisPosition"
{ S7_Optimized_Access := 'FALSE' }
VERSION : 0.1
   VAR_INPUT 
      "Sensor Controlled" : Bool;
      Axis_Sensor_On_Position : Bool;
      Axis_Encoder_On_Position : Bool;
   END_VAR

   VAR_OUTPUT 
      Axis_Measuring_Mode : Bool;
   END_VAR


BEGIN
	IF #"Sensor Controlled" THEN
	    #Axis_Measuring_Mode := #Axis_Sensor_On_Position;
	ELSE
	    #Axis_Measuring_Mode := #Axis_Encoder_On_Position;
	END_IF;
	
END_FUNCTION_BLOCK

FUNCTION_BLOCK "DriveConfirmation_Function"   // FB5, FBD
TITLE = Drive Confirmation Function Block
VERSION : 0.1
// stored: AutoNumber true, IsIECCheckEnabled false, UDAEnableTagReadback false
   VAR_INPUT
      "System RUN" : Bool;
      "Drive Ouput Q" : Bool;
      "Drive Ready Signal" : Bool;
      DelayTime : Time := T#1s;
   END_VAR
   VAR_OUTPUT
      "Timer ET" : Time;
      "Ouput WORD" : Bool;
   END_VAR
BEGIN

REGION Network 1: Confirmation Drive
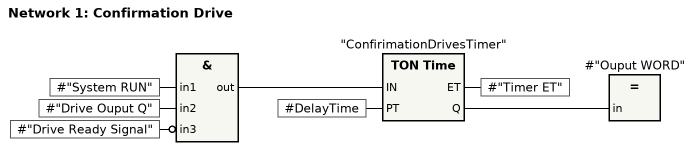
   "ConfirimationDrivesTimer".TON(IN := #"System RUN" AND #"Drive Ouput Q" AND NOT #"Drive Ready Signal",
                           PT := #DelayTime,
                           ET => #"Timer ET");
   #"Ouput WORD" := "ConfirimationDrivesTimer".Q;
END_REGION
END_FUNCTION_BLOCK

FUNCTION "9 - OVERIG" : Void   // FC6, LAD
TITLE = Other - Testing
VERSION : 0.1
// stored: AutoNumber true, IsIECCheckEnabled false, UDAEnableTagReadback false
   VAR_TEMP
      Encoder : Int;
      Gate : Bool;
      GATESTP : Bool;
      OTERRA : Bool;
      Direct : Bool;
      Prepar : Bool;
      CMPV1 : Bool;
      CMPV2 : Bool;
      RESSYNC : Bool;
      RESZERO : Bool;
      OTERR : Bool;
   END_VAR
BEGIN

REGION Network 1: SAFETY - OVERRIDE
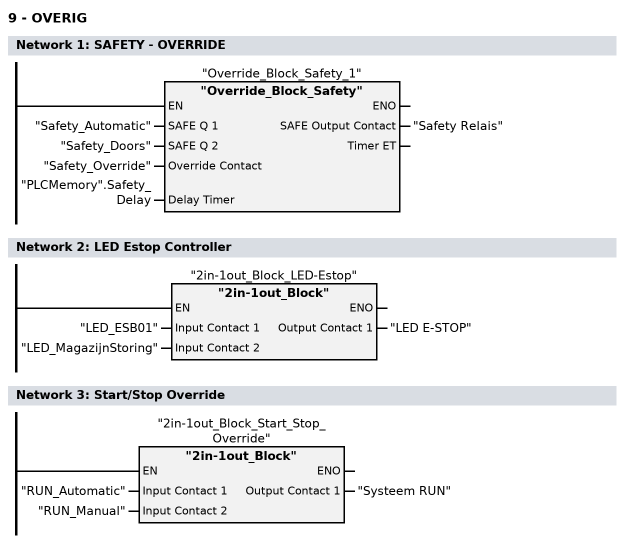
   RUNG wire#powerrail
      "Override_Block_Safety_1"("SAFE Q 1" := "Safety_Automatic", "SAFE Q 2" := "Safety_Doors", "Override Contact" := "Safety_Override", "Delay Timer" := "PLCMemory".Safety_Delay, "SAFE Output Contact" => "Safety Relais", "Timer ET" =>)
   END_RUNG
   // the same network as SCL:
   "Override_Block_Safety_1"("SAFE Q 1" := "Safety_Automatic",   // "Override_Block_Safety"
                           "SAFE Q 2" := "Safety_Doors",
                           "Override Contact" := "Safety_Override",
                           "Delay Timer" := "PLCMemory".Safety_Delay,
                           "SAFE Output Contact" => "Safety Relais");
END_REGION

REGION Network 2: LED Estop Controller
   RUNG wire#powerrail
      "2in-1out_Block_LED-Estop"("Input Contact 1" := "LED_ESB01", "Input Contact 2" := "LED_MagazijnStoring", "Output Contact 1" => "LED E-STOP")
   END_RUNG
   // the same network as SCL:
   "2in-1out_Block_LED-Estop"("Input Contact 1" := "LED_ESB01",   // "2in-1out_Block"
                           "Input Contact 2" := "LED_MagazijnStoring",
                           "Output Contact 1" => "LED E-STOP");
END_REGION

REGION Network 3: Start/Stop Override
   RUNG wire#powerrail
      "2in-1out_Block_Start_Stop_Override"("Input Contact 1" := "RUN_Automatic", "Input Contact 2" := "RUN_Manual", "Output Contact 1" => "Systeem RUN")
   END_RUNG
   // the same network as SCL:
   "2in-1out_Block_Start_Stop_Override"("Input Contact 1" := "RUN_Automatic",   // "2in-1out_Block"
                           "Input Contact 2" := "RUN_Manual",
                           "Output Contact 1" => "Systeem RUN");
END_REGION
END_FUNCTION

FUNCTION_BLOCK "Override_Block_Safety"   // FB7, FBD
TITLE = Override Block Safety.
VERSION : 0.1
// stored: AutoNumber true, IsIECCheckEnabled false, UDAEnableTagReadback false
   VAR_INPUT
      "SAFE Q 1" : Bool;
      "SAFE Q 2" : Bool;
      "Override Contact" : Bool;
      "Delay Timer" : Time;
   END_VAR
   VAR_OUTPUT
      "SAFE Output Contact" : Bool;
      "Timer ET" : Time;
   END_VAR
BEGIN

REGION Network 1: SAFETY - OVERRIDE
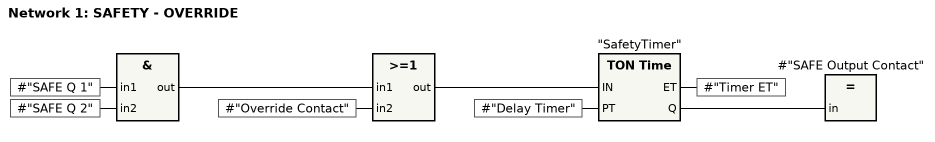
   "SafetyTimer".TON(IN := (#"SAFE Q 1" AND #"SAFE Q 2") OR #"Override Contact",
                     PT := #"Delay Timer",
                     ET => #"Timer ET");
   #"SAFE Output Contact" := "SafetyTimer".Q;
END_REGION
END_FUNCTION_BLOCK

FUNCTION_BLOCK "2in-1out_Block"   // FB6, FBD
VERSION : 0.1
// stored: AutoNumber true, IsIECCheckEnabled true, UDAEnableTagReadback false
   VAR_INPUT
      "Input Contact 1" : Bool;
      "Input Contact 2" : Bool;
   END_VAR
   VAR_OUTPUT
      "Output Contact 1" : Bool;
   END_VAR
BEGIN

REGION Network 1: Network Default
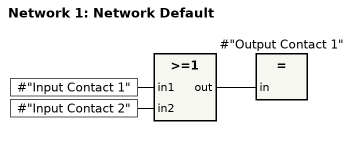
   #"Output Contact 1" := #"Input Contact 1" OR #"Input Contact 2";
END_REGION
END_FUNCTION_BLOCK

FUNCTION_BLOCK "ResetOuputs_Function"   // FB9, LAD
TITLE = Reset Ouput Functions With Commands
VERSION : 0.1
// stored: AutoNumber true, IsIECCheckEnabled false, UDAEnableTagReadback false
   VAR_INPUT
      StopCommand_NC : Bool;
      StopCommand_NO : Bool;
   END_VAR
   VAR_OUTPUT
      Output_1 : Bool;
      Output_2 : Bool;
      Output_3 : Bool;
      Output_4 : Bool;
      Output_5 : Bool;
      Output_6 : Bool;
      Output_7 : Bool;
      Output_8 : Bool;
      Output_9 : Bool;
      Output_10 : Bool;
   END_VAR
BEGIN

REGION Network 1: NW1
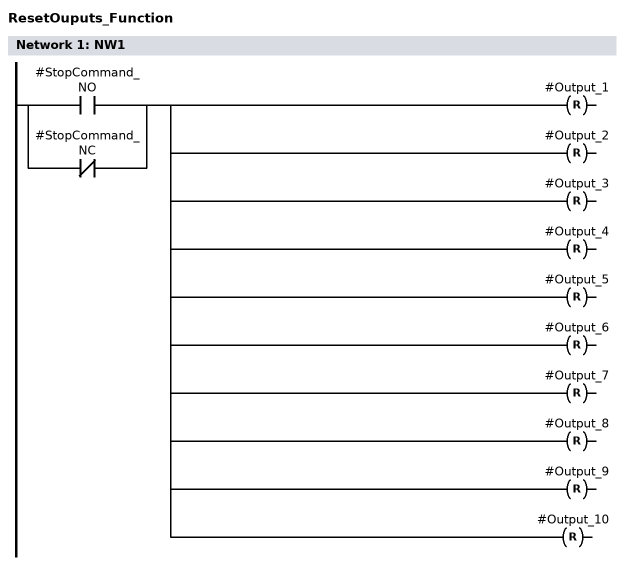
   RUNG wire#powerrail
      Contact( #StopCommand_NO )
      wire#w1
      R_Coil( #Output_1 )
   END_RUNG
   RUNG wire#powerrail
      I_Contact( #StopCommand_NC )
   END_RUNG wire#w1
   RUNG wire#w1
      R_Coil( #Output_2 )
   END_RUNG
   RUNG wire#w1
      R_Coil( #Output_3 )
   END_RUNG
   RUNG wire#w1
      R_Coil( #Output_4 )
   END_RUNG
   RUNG wire#w1
      R_Coil( #Output_5 )
   END_RUNG
   RUNG wire#w1
      R_Coil( #Output_6 )
   END_RUNG
   RUNG wire#w1
      R_Coil( #Output_7 )
   END_RUNG
   RUNG wire#w1
      R_Coil( #Output_8 )
   END_RUNG
   RUNG wire#w1
      R_Coil( #Output_9 )
   END_RUNG
   RUNG wire#w1
      R_Coil( #Output_10 )
   END_RUNG
   // the same network as SCL:
   IF #StopCommand_NO OR NOT #StopCommand_NC THEN
       #Output_1 := FALSE;
       #Output_2 := FALSE;
       #Output_3 := FALSE;
       #Output_4 := FALSE;
       #Output_5 := FALSE;
       #Output_6 := FALSE;
       #Output_7 := FALSE;
       #Output_8 := FALSE;
       #Output_9 := FALSE;
       #Output_10 := FALSE;
   END_IF;
END_REGION
END_FUNCTION_BLOCK

FUNCTION "SCL_Block" : Void
{ S7_Optimized_Access := 'FALSE' }
VERSION : 0.1

BEGIN
	// Reset de Word variabelen aan het begin van elke cyclus
	"Alarms".AlarmsWord := 0;
	"Alarms".HMI_Alarm_Drive1 := 0;
	"Alarms".HMI_Alarm_Drive2 := 0;
	"Alarms".HMI_Alarm_Drive3 := 0;
	"Alarms".HMI_Alarm_Drive4 := 0;
	"Alarms".HMI_Alarm_Drive5 := 0;
	
	// Controleer de alarmen en zet de respectievelijke bits aan
	IF "Alarms".AlarmStruct.Alarm_Product_Not_Position THEN
	    "Alarms".AlarmsWord := "Alarms".AlarmsWord OR WORD#1; // Zet bit 0 aan
	END_IF;
	
	IF "Alarms".AlarmStruct.Alarm_Axis_Not_Position THEN
	    "Alarms".AlarmsWord := "Alarms".AlarmsWord OR WORD#2; // Zet bit 1 aan
	END_IF;
	
	IF "Alarms".AlarmStruct.Alarm_Drive1 THEN
	    "Alarms".HMI_Alarm_Drive1 := "Alarms".HMI_Alarm_Drive1 OR WORD#1; // Zet bit 2 aan
	END_IF;
	
	IF "Alarms".AlarmStruct.Alarm_Drive2 THEN
	    "Alarms".HMI_Alarm_Drive2 := "Alarms".HMI_Alarm_Drive2 OR WORD#1; // Zet bit 3 aan
	END_IF;
	
	IF "Alarms".AlarmStruct.Alarm_Drive3 THEN
	    "Alarms".HMI_Alarm_Drive3 := "Alarms".HMI_Alarm_Drive3 OR WORD#1; // Zet bit 4 aan
	END_IF;
	
	IF "Alarms".AlarmStruct.Alarm_Drive4 THEN
	    "Alarms".HMI_Alarm_Drive4 := "Alarms".HMI_Alarm_Drive4 OR WORD#1; // Zet bit 5 aan
	END_IF;
	
	IF "Alarms".AlarmStruct.Alarm_Drive5 THEN
	    "Alarms".HMI_Alarm_Drive5 := "Alarms".HMI_Alarm_Drive5 OR WORD#1; // Zet bit 6 aan
	END_IF;
	
	
	// Position Program Axis 3 (Wals)
	
	// Configureer de timer om elke 0,5 seconde af te lopen
	"Timer_0_5s".TON(IN := TRUE,
	PT := "PLCMemory"."Encoder PulsOffset");
	
	// Controleer of de timer is afgelopen
	IF "Timer_0_5s".Q THEN
	    // Verhoog of verlaag de positie afhankelijk van de aandrijfsignalen
	    IF "Drive 3 RUN FWD" THEN
	        "PLCMemory".EncoderPosition := "PLCMemory".EncoderPosition + "PLCMemory".StepSize; // Verhoog met de stepgrootte
	    ELSIF "Drive 3 REV" THEN
	        "PLCMemory".EncoderPosition := "PLCMemory".EncoderPosition - "PLCMemory".StepSize; // Verlaag met de stepgrootte
	    END_IF;
	    
	    // Wrapping van de positie bij overschrijden van 360 graden of onder 0 graden
	    IF "PLCMemory".EncoderPosition >= 360.0 THEN
	        "PLCMemory".EncoderPosition := 0.0;  // Wrapping naar 0 als de positie 360 overschrijdt
	    ELSIF "PLCMemory".EncoderPosition < 0.0 THEN
	        "PLCMemory".EncoderPosition := 360.0; // Wrapping naar 360 als de positie onder 0 gaat
	    END_IF;
	    
	    // Reset de timer
	    "Timer_0_5s".TON (IN := FALSE,
	                      PT := "PLCMemory"."Encoder PulsOffset"); // Reset de timer zodat deze opnieuw kan starten
	END_IF;
	
	// Homing logica
	IF "Sensor Wals (Option)" THEN
	    "PLCMemory".EncoderPosition := 0.0;  // Reset de positie naar 0 als de sensor wordt geactiveerd
	END_IF;
	
	
	
	//Drive Servo Control Here:
	/// Desired Position Axis 3
	
	// Controleer of de HMI-knop is ingedrukt en er een gewenste positie is ingesteld
	//IF "HMI_Des_Pos_Axis3" THEN
	    //"GoButtonPressed" := TRUE; // HMI-knop is ingedrukt, start beweging
	//END_IF;
	
	// Beveiliging voor de Desired_Encoder_Position: Zorg dat de waarde tussen 0 en 360 blijft
	//IF "PLCMemory".Desired_Encoder_Position > 360.0 THEN
	  //  "PLCMemory".Desired_Encoder_Position := 360.0;  // Zet naar 360 als de waarde boven 360 ligt
	//ELSIF "PLCMemory".Desired_Encoder_Position < 0.0 THEN
	    //"PLCMemory".Desired_Encoder_Position := 0.0;  // Zet naar 0 als de waarde onder 0 ligt
	//END_IF;
	
	// Wrapping van de gewenste positie: Als de gewenste positie 360 is, zet deze dan op 0
	//IF "PLCMemory".Desired_Encoder_Position = 360.0 THEN
	   // "PLCMemory".Desired_Encoder_Position := 0.0;  // Wrapping naar 0 als de gewenste positie 360 is
	//END_IF;
	
	// Voer beweging uit totdat de gewenste positie is bereikt
	//IF "GoButtonPressed" THEN
	    // Bepaal de bewegingsrichting en start de beweging
	  //  IF "PLCMemory".EncoderPosition < "PLCMemory".Desired_Encoder_Position - "PLCMemory".Tolerance THEN
	        // Beweeg vooruit met StepSize als snelheid
	      //  "PLCMemory".EncoderPosition := "PLCMemory".EncoderPosition + "PLCMemory".StepSize;
	     //   "Drive_3_Manual" := TRUE;   // Activeer vooruitbeweging
	      //  "Drive 3 REV" := FALSE;     // Zorg dat achteruitbeweging uit is
	        
	  //  ELSIF "PLCMemory".EncoderPosition > "PLCMemory".Desired_Encoder_Position + "PLCMemory".Tolerance THEN
	        // Beweeg achteruit met StepSize als snelheid
	     //   "PLCMemory".EncoderPosition := "PLCMemory".EncoderPosition - "PLCMemory".StepSize;
	    //    "Drive_3_Manual" := FALSE;  // Zorg dat vooruitbeweging uit is
	    //    "Drive 3 REV" := TRUE;      // Activeer achteruitbeweging
	        
	   // ELSE
	        // Stop de beweging zodra de positie binnen de tolerantie komt
	      //  "Drive_3_Manual" := FALSE;    // Zet vooruitbeweging uit
	     //   "Drive 3 REV" := FALSE;       // Zet achteruitbeweging uit
	     //   "GoButtonPressed" := FALSE;   // Zet de Go-knop uit om verdere beweging te stoppen
	   // END_IF;
	//END_IF;
	
	
	
	
	
END_FUNCTION

FUNCTION "7 - Clean" : Void   // FC4, LAD
TITLE = Cleaning Program
VERSION : 0.1
// stored: AutoNumber true, IsIECCheckEnabled false, UDAEnableTagReadback false
   VAR_TEMP
      BlowOff_Active : Bool;
   END_VAR
   VAR_TEMP   // added for the SCL form of the ladder/FBD networks
      _w1 : Bool;
   END_VAR
BEGIN

REGION Network 1: Button Pressed Show Message
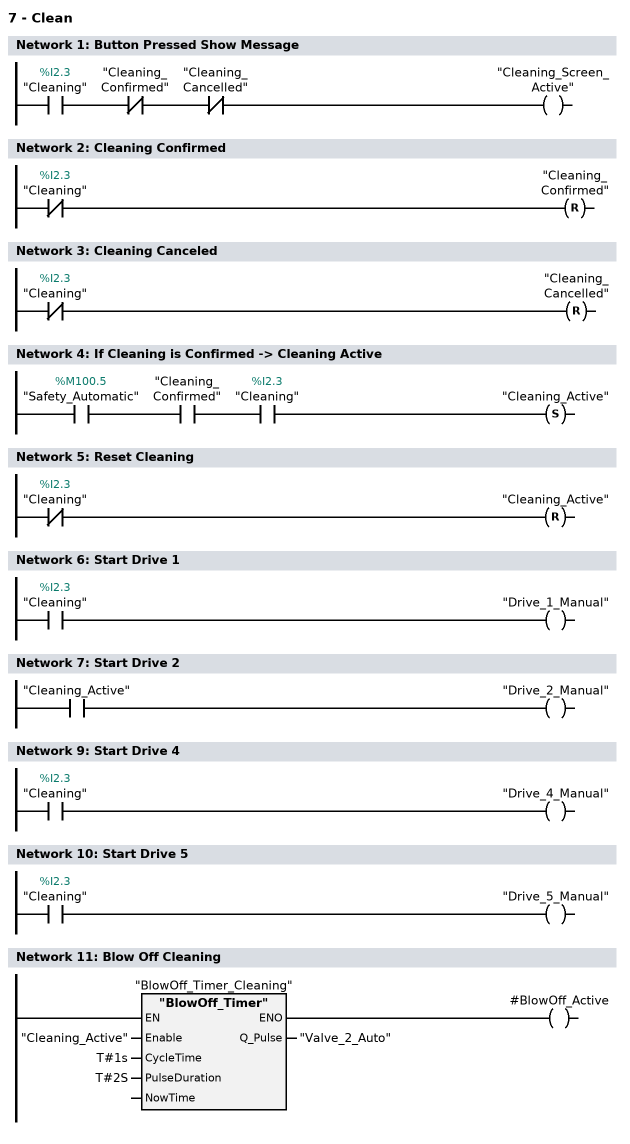
   RUNG wire#powerrail
      Contact( "Cleaning" )
      I_Contact( "Cleaning_Confirmed" )
      I_Contact( "Cleaning_Cancelled" )
      Coil( "Cleaning_Screen_Active" )
   END_RUNG
   // the same network as SCL:
   "Cleaning_Screen_Active" := "Cleaning" AND NOT "Cleaning_Confirmed" AND NOT "Cleaning_Cancelled";
END_REGION

REGION Network 2: Cleaning Confirmed
   RUNG wire#powerrail
      I_Contact( "Cleaning" )
      R_Coil( "Cleaning_Confirmed" )
   END_RUNG
   // the same network as SCL:
   IF NOT "Cleaning" THEN "Cleaning_Confirmed" := FALSE; END_IF;
END_REGION

REGION Network 3: Cleaning Canceled
   RUNG wire#powerrail
      I_Contact( "Cleaning" )
      R_Coil( "Cleaning_Cancelled" )
   END_RUNG
   // the same network as SCL:
   IF NOT "Cleaning" THEN "Cleaning_Cancelled" := FALSE; END_IF;
END_REGION

REGION Network 4: If Cleaning is Confirmed -> Cleaning Active
   RUNG wire#powerrail
      Contact( "Safety_Automatic" )
      Contact( "Cleaning_Confirmed" )
      Contact( "Cleaning" )
      S_Coil( "Cleaning_Active" )
   END_RUNG
   // the same network as SCL:
   IF "Safety_Automatic" AND "Cleaning_Confirmed" AND "Cleaning" THEN "Cleaning_Active" := TRUE; END_IF;
END_REGION

REGION Network 5: Reset Cleaning
   RUNG wire#powerrail
      I_Contact( "Cleaning" )
      R_Coil( "Cleaning_Active" )
   END_RUNG
   // the same network as SCL:
   IF NOT "Cleaning" THEN "Cleaning_Active" := FALSE; END_IF;
END_REGION

REGION Network 6: Start Drive 1
   RUNG wire#powerrail
      Contact( "Cleaning" )
      Coil( "Drive_1_Manual" )
   END_RUNG
   // the same network as SCL:
   "Drive_1_Manual" := "Cleaning";
END_REGION

REGION Network 7: Start Drive 2
   RUNG wire#powerrail
      Contact( "Cleaning_Active" )
      Coil( "Drive_2_Manual" )
   END_RUNG
   // the same network as SCL:
   "Drive_2_Manual" := "Cleaning_Active";
END_REGION

REGION Network 8: Start Drive 3
END_REGION

REGION Network 9: Start Drive 4
   RUNG wire#powerrail
      Contact( "Cleaning" )
      Coil( "Drive_4_Manual" )
   END_RUNG
   // the same network as SCL:
   "Drive_4_Manual" := "Cleaning";
END_REGION

REGION Network 10: Start Drive 5
   RUNG wire#powerrail
      Contact( "Cleaning" )
      Coil( "Drive_5_Manual" )
   END_RUNG
   // the same network as SCL:
   "Drive_5_Manual" := "Cleaning";
END_REGION

REGION Network 11: Blow Off Cleaning
   RUNG wire#powerrail
      "BlowOff_Timer_Cleaning"(Enable := "Cleaning_Active", CycleTime := T#1s, PulseDuration := T#2S, Q_Pulse => "Valve_2_Auto", NowTime :=)
      Coil( #BlowOff_Active )
   END_RUNG
   // the same network as SCL:
   "BlowOff_Timer_Cleaning"(Enable := "Cleaning_Active",   // "BlowOff_Timer"
                           CycleTime := T#1s,
                           PulseDuration := T#2S,
                           Q_Pulse => "Valve_2_Auto",
                           ENO => #_w1);
   #BlowOff_Active := #_w1;
END_REGION
END_FUNCTION

FUNCTION "Servo_DriveManager" : Void   // FC17, FBD
TITLE = Drive Manager Closed Loop
VERSION : 0.1
// Drive Manager for Closed Loop with Encoder
// stored: AutoNumber true, IsIECCheckEnabled false, UDAEnableTagReadback false
   VAR_INPUT
      "[NAME] Axis Name" : String;
      "[INPUT] ReferenceSwitch_Input" : Bool;
      "[INPUT] Drive Ready" : Bool;
      "[INPUT] E-STOP Check" : Bool;
      "[COMMAND] Start_Reference Run" : Bool;
      "[COMMAND] Take_over_Pos" : Bool;
      "[COMMAND] Go to Position" : Bool;
      "[COMMAND] Axis Manual Forward" : Bool;
      "[COMMAND] Axis Manual Reverse" : Bool;
      "[COMMAND] Axis Speed" : Int;
      "[COMMAND] Axis Fast Stop" : Bool;
      "[COMMAND] Go To Rest" : Bool;
      "[COMMAND] Axis Brake" : Bool;
      "[VALUE] Reference Position" : Int;
      "[VALUE] Set Position" : Real;
      "[VALUE] Rest Position" : Real;
      "[VALUE] Accelerating" : Real;
      "[VALUE] Deaccelerating" : Real;
      "[VALUE] Position Tolerance" : Real;
      "[COMMUNICATION] MasterWord" : String;
      "[COMMUNICATION] Callback" : String;
   END_VAR
   VAR_OUTPUT
      "[OUTPUT] Drive FWD Command" : Bool;
      "[OUTPUT] Drive REV Command" : Bool;
      "[OUTPUT] Drive Speed 2 (50%)" : Bool;
      "[OUTPUT] Drive Speed 3 (75%)" : Bool;
      "[OUTPUT] Drive Fast Stop Command" : Bool;
      "[MESSAGE] Axis Busy" : Bool;
      "[MESSAGE] Error Executing" : Bool;
      "[MESSAGE] Axis On Position" : Bool;
      "[MESSAGE] Axis On Rest" : Bool;
      "[MESSAGE] Drive State" : String;
      "[MESSAGE] Axis Slips" : String;
   END_VAR
   VAR_TEMP
      UnscPos : Int;
      ScPos : Real;
      ActEncPos : Real;
      SetRefRun : Bool;
      SetRefRun_Q : Bool;
      MoveToRest : Bool;
      MoveToRest_Q : Bool;
      Automatic_Positive : Bool;
      Manual_Positive : Bool;
      Automatic_Negative : Bool;
      Manual_Negative : Bool;
      HS_Positive : Bool;
      MasterWordHex : Int;
      Speed50 : Bool;
      Speed75 : Bool;
      Min_Position : Real;
      Max_Position : Real;
      Axis_On_Position : Bool;
      Direction_Forward : Bool;
      Direction_Backward : Bool;
      Drive_Auto_Fwd : Bool;
      InternalFastStop : Bool;
      RefRunSetSignal : Bool;
      GoToRest2 : Bool;
      "[COMMAND] Go to Position_Rest" : Bool;
      RestPos_SpareMove : Real;
   END_VAR
   VAR_TEMP   // added for the SCL form of the ladder/FBD networks
      _w1 : Bool;
   END_VAR
BEGIN

REGION Network 1: Reference Run
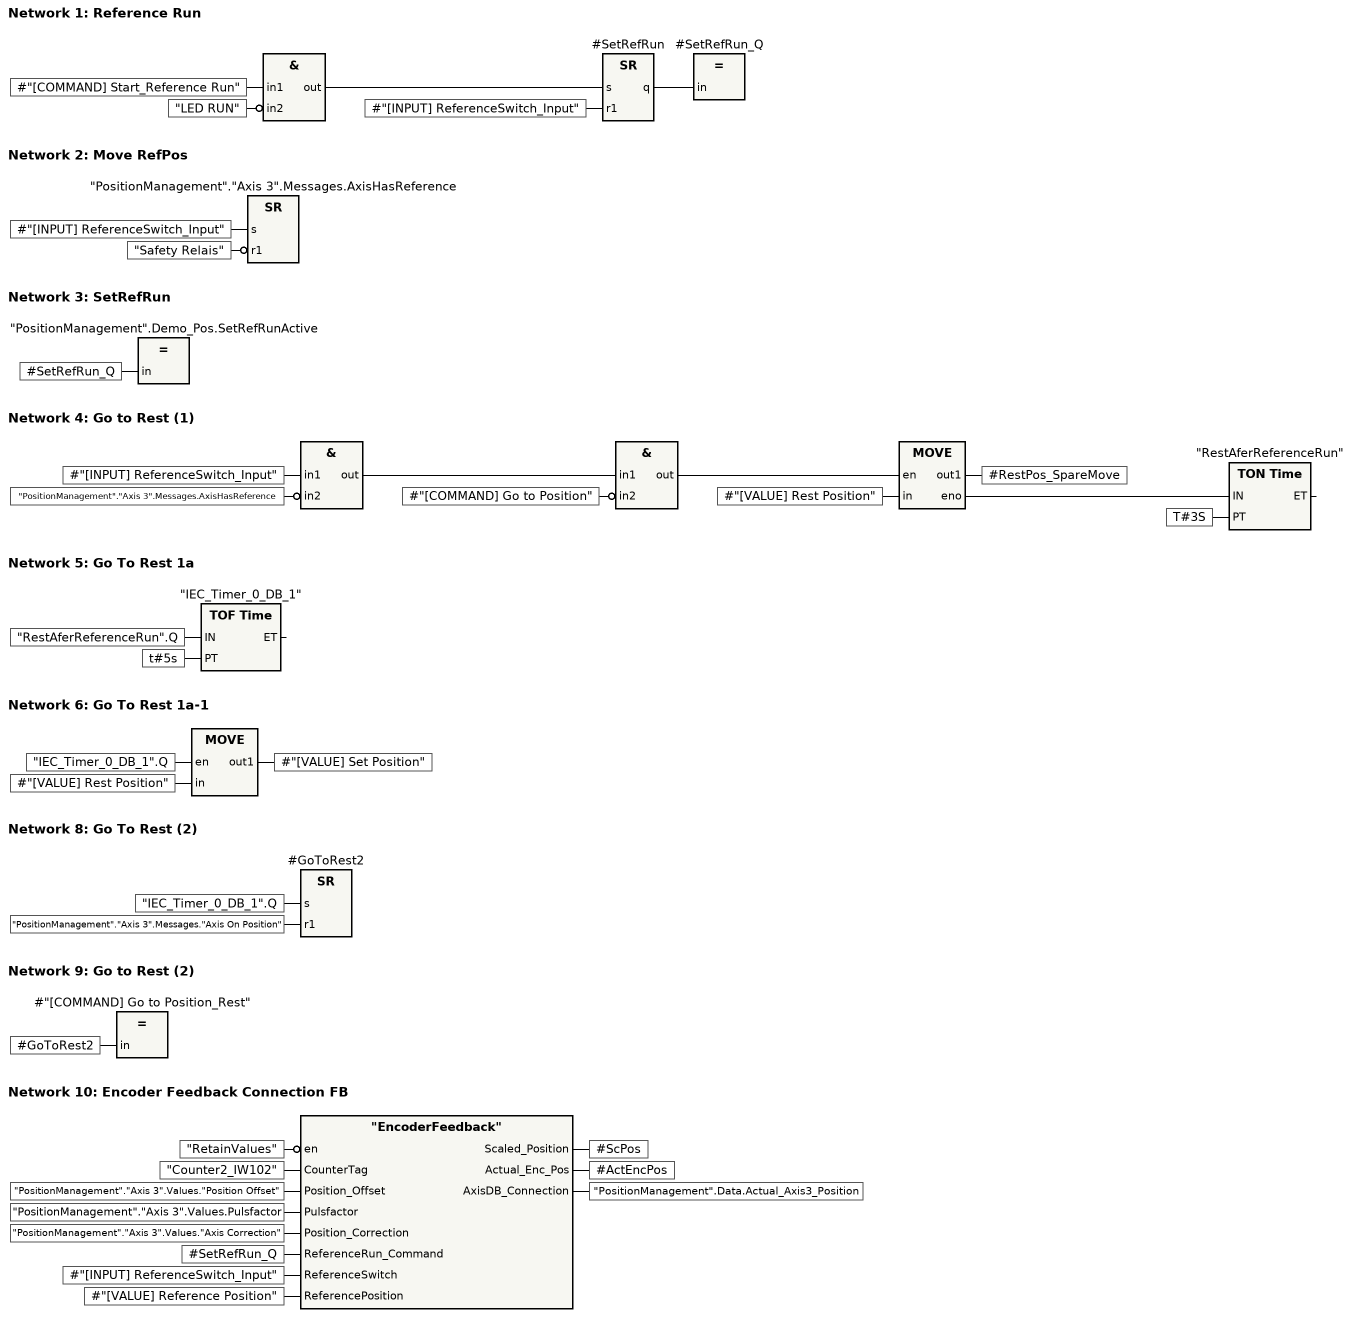
   IF #"[COMMAND] Start_Reference Run" AND NOT "LED RUN" THEN
       #SetRefRun := TRUE;   // SR flip-flop
   END_IF;
   IF #"[INPUT] ReferenceSwitch_Input" THEN #SetRefRun := FALSE; END_IF;
   #SetRefRun_Q := #SetRefRun;
END_REGION

REGION Network 2: Move RefPos
   IF #"[INPUT] ReferenceSwitch_Input" THEN
       "PositionManagement"."Axis 3".Messages.AxisHasReference := TRUE;   // SR flip-flop
   END_IF;
   IF NOT "Safety Relais" THEN "PositionManagement"."Axis 3".Messages.AxisHasReference := FALSE; END_IF;
END_REGION

REGION Network 3: SetRefRun
   "PositionManagement".Demo_Pos.SetRefRunActive := #SetRefRun_Q;
END_REGION

REGION Network 4: Go to Rest (1)
   // ENO of a box is taken as its EN; it also drops when the box reports an error
   #_w1 := #"[INPUT] ReferenceSwitch_Input" AND NOT "PositionManagement"."Axis 3".Messages.AxisHasReference AND NOT #"[COMMAND] Go to Position";
   IF #_w1 THEN #RestPos_SpareMove := #"[VALUE] Rest Position"; END_IF;
   "RestAferReferenceRun".TON(IN := #_w1, PT := T#3S);
END_REGION

REGION Network 5: Go To Rest 1a
   "IEC_Timer_0_DB_1".TOF(IN := "RestAferReferenceRun".Q, PT := t#5s);
END_REGION

REGION Network 6: Go To Rest 1a-1
   IF "IEC_Timer_0_DB_1".Q THEN #"[VALUE] Set Position" := #"[VALUE] Rest Position"; END_IF;
END_REGION

REGION Network 7: Go To Rest 1b
END_REGION

REGION Network 8: Go To Rest (2)
   IF "IEC_Timer_0_DB_1".Q THEN
       #GoToRest2 := TRUE;   // SR flip-flop
   END_IF;
   IF "PositionManagement"."Axis 3".Messages."Axis On Position" THEN #GoToRest2 := FALSE; END_IF;
END_REGION

REGION Network 9: Go to Rest (2)
   #"[COMMAND] Go to Position_Rest" := #GoToRest2;
END_REGION

REGION Network 10: Encoder Feedback Connection FB
   // Getting the feedback from the encoder device
   IF NOT "RetainValues" THEN
       "EncoderFeedback"(CounterTag := "Counter2_IW102",
                         Position_Offset := "PositionManagement"."Axis 3".Values."Position Offset",
                         Pulsfactor := "PositionManagement"."Axis 3".Values.Pulsfactor,
                         Position_Correction := "PositionManagement"."Axis 3".Values."Axis Correction",
                         ReferenceRun_Command := #SetRefRun_Q,
                         ReferenceSwitch := #"[INPUT] ReferenceSwitch_Input",
                         ReferencePosition := #"[VALUE] Reference Position",
                         Scaled_Position => #ScPos,
                         Actual_Enc_Pos => #ActEncPos,
                         AxisDB_Connection => "PositionManagement".Data.Actual_Axis3_Position);
   END_IF;
END_REGION

REGION Network 11: Calculate Position Tolerance 1
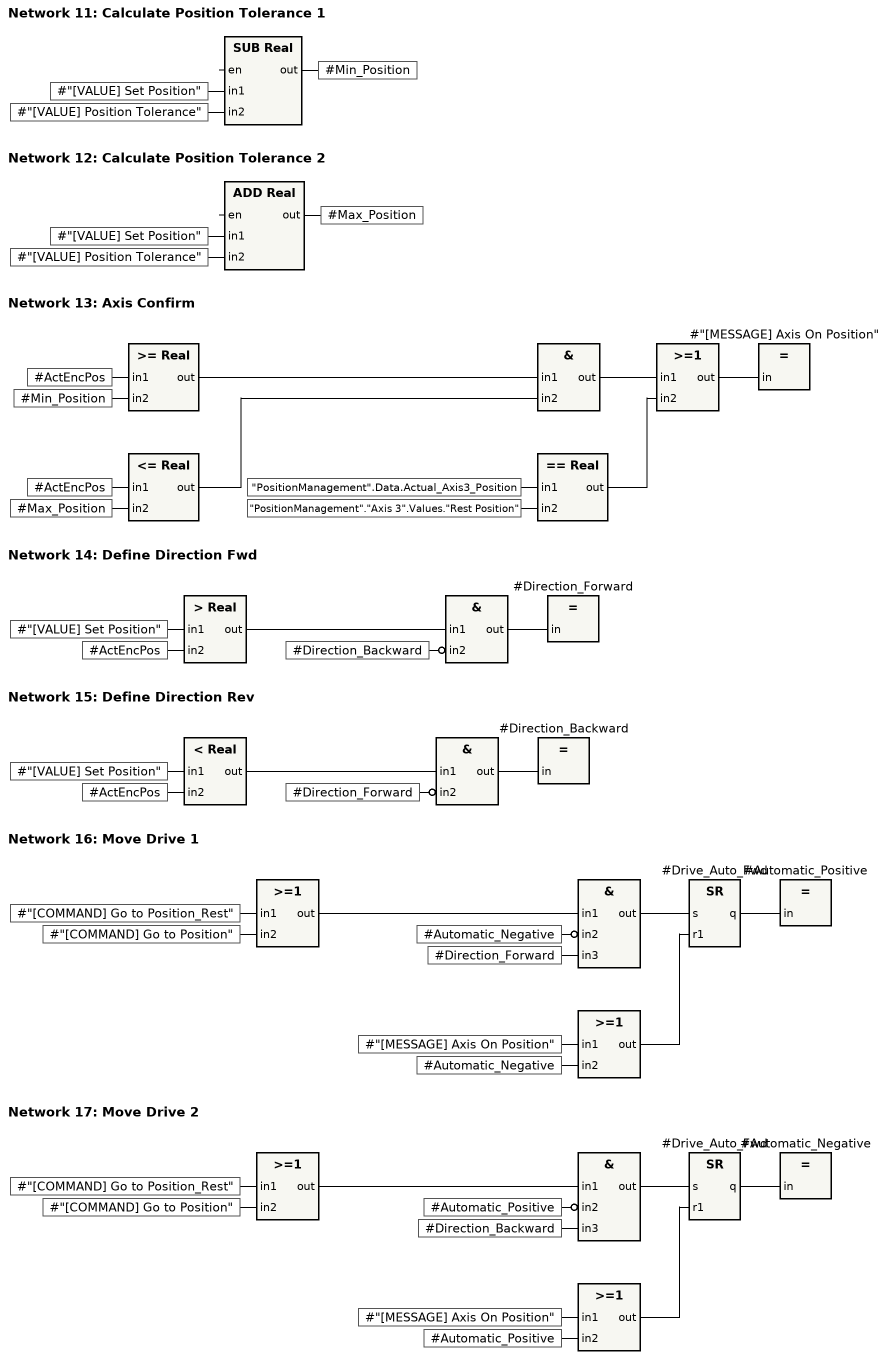
   #Min_Position := #"[VALUE] Set Position" - #"[VALUE] Position Tolerance";
END_REGION

REGION Network 12: Calculate Position Tolerance 2
   #Max_Position := #"[VALUE] Set Position" + #"[VALUE] Position Tolerance";
END_REGION

REGION Network 13: Axis Confirm
   #"[MESSAGE] Axis On Position" := ((#ActEncPos >= #Min_Position) AND (#ActEncPos <= #Max_Position)) OR ("PositionManagement".Data.Actual_Axis3_Position = "PositionManagement"."Axis 3".Values."Rest Position");
END_REGION

REGION Network 14: Define Direction Fwd
   #Direction_Forward := (#"[VALUE] Set Position" > #ActEncPos) AND NOT #Direction_Backward;
END_REGION

REGION Network 15: Define Direction Rev
   #Direction_Backward := (#"[VALUE] Set Position" < #ActEncPos) AND NOT #Direction_Forward;
END_REGION

REGION Network 16: Move Drive 1
   IF (#"[COMMAND] Go to Position_Rest" OR #"[COMMAND] Go to Position") AND NOT #Automatic_Negative AND #Direction_Forward THEN
       #Drive_Auto_Fwd := TRUE;   // SR flip-flop
   END_IF;
   IF #"[MESSAGE] Axis On Position" OR #Automatic_Negative THEN #Drive_Auto_Fwd := FALSE; END_IF;
   #Automatic_Positive := #Drive_Auto_Fwd;
END_REGION

REGION Network 17: Move Drive 2
   IF (#"[COMMAND] Go to Position_Rest" OR #"[COMMAND] Go to Position") AND NOT #Automatic_Positive AND #Direction_Backward THEN
       #Drive_Auto_Fwd := TRUE;   // SR flip-flop
   END_IF;
   IF #"[MESSAGE] Axis On Position" OR #Automatic_Positive THEN #Drive_Auto_Fwd := FALSE; END_IF;
   #Automatic_Negative := #Drive_Auto_Fwd;
END_REGION

REGION Network 18: Manual Displacement Positive
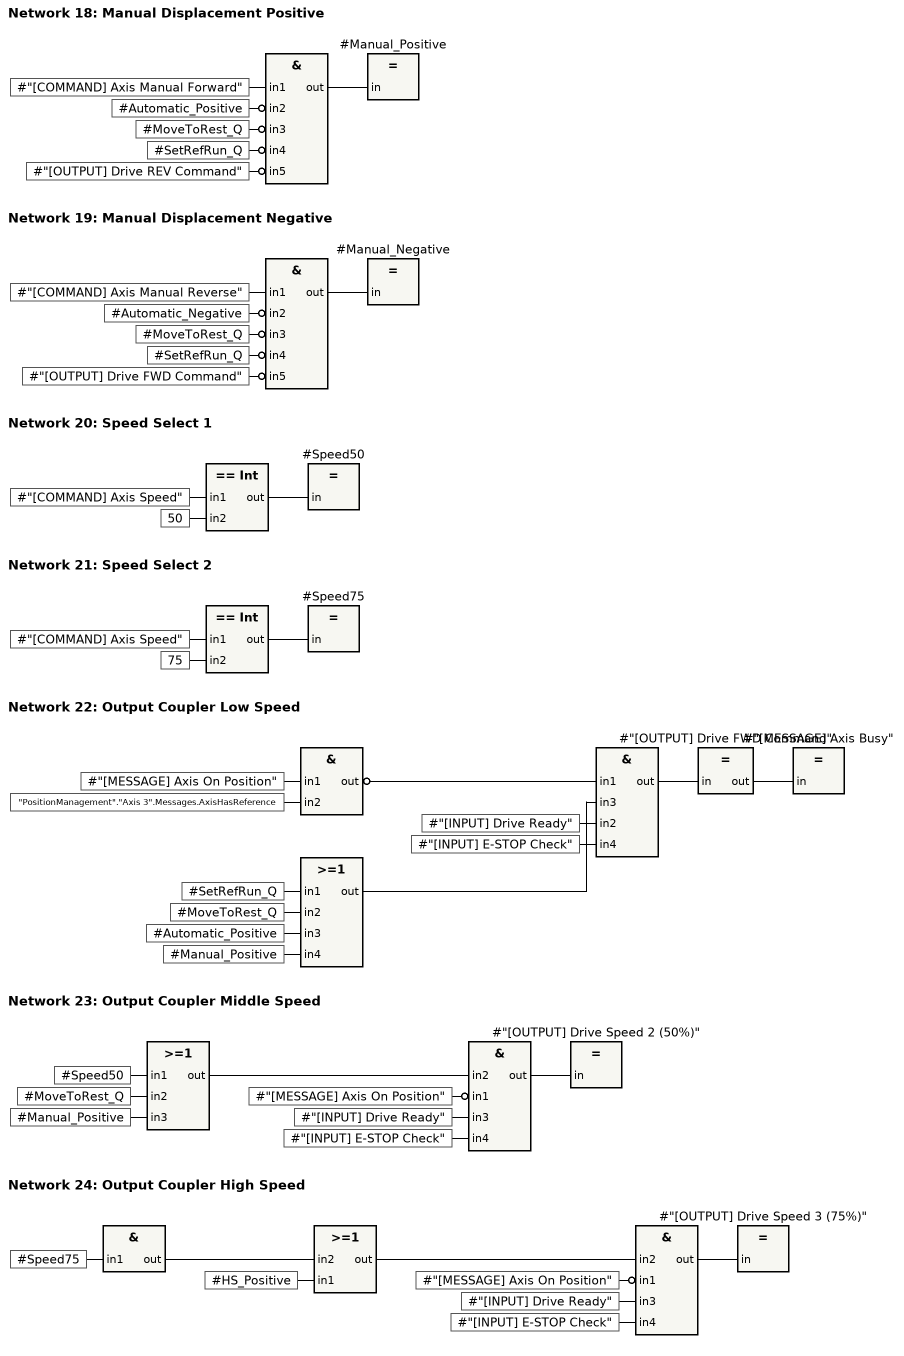
   #Manual_Positive := #"[COMMAND] Axis Manual Forward" AND NOT #Automatic_Positive AND NOT #MoveToRest_Q AND NOT #SetRefRun_Q AND NOT #"[OUTPUT] Drive REV Command";
END_REGION

REGION Network 19: Manual Displacement Negative
   #Manual_Negative := #"[COMMAND] Axis Manual Reverse" AND NOT #Automatic_Negative AND NOT #MoveToRest_Q AND NOT #SetRefRun_Q AND NOT #"[OUTPUT] Drive FWD Command";
END_REGION

REGION Network 20: Speed Select 1
   #Speed50 := #"[COMMAND] Axis Speed" = 50;
END_REGION

REGION Network 21: Speed Select 2
   #Speed75 := #"[COMMAND] Axis Speed" = 75;
END_REGION

REGION Network 22: Output Coupler Low Speed
   #_w1 := NOT (#"[MESSAGE] Axis On Position" AND "PositionManagement"."Axis 3".Messages.AxisHasReference) AND (#SetRefRun_Q OR #MoveToRest_Q OR #Automatic_Positive OR #Manual_Positive) AND #"[INPUT] Drive Ready" AND #"[INPUT] E-STOP Check";
   #"[OUTPUT] Drive FWD Command" := #_w1;
   #"[MESSAGE] Axis Busy" := #_w1;
END_REGION

REGION Network 23: Output Coupler Middle Speed
   #"[OUTPUT] Drive Speed 2 (50%)" := (#Speed50 OR #MoveToRest_Q OR #Manual_Positive) AND NOT #"[MESSAGE] Axis On Position" AND #"[INPUT] Drive Ready" AND #"[INPUT] E-STOP Check";
END_REGION

REGION Network 24: Output Coupler High Speed
   #"[OUTPUT] Drive Speed 3 (75%)" := (#Speed75 OR #HS_Positive) AND NOT #"[MESSAGE] Axis On Position" AND #"[INPUT] Drive Ready" AND #"[INPUT] E-STOP Check";
END_REGION

REGION Network 25: Output Coupler Reverse
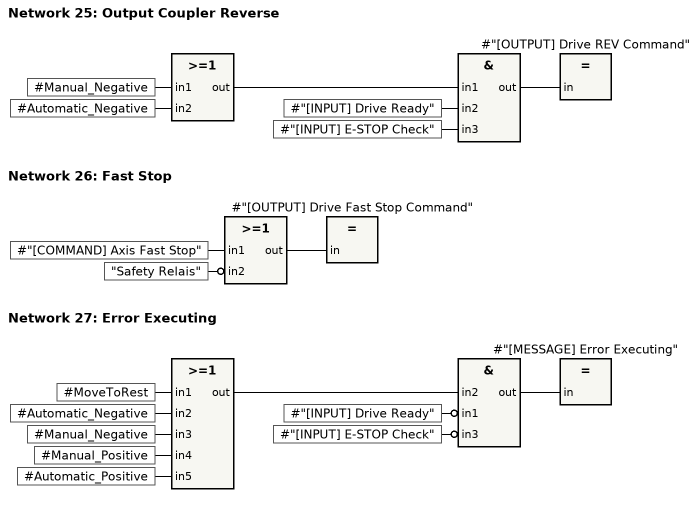
   #"[OUTPUT] Drive REV Command" := (#Manual_Negative OR #Automatic_Negative) AND #"[INPUT] Drive Ready" AND #"[INPUT] E-STOP Check";
END_REGION

REGION Network 26: Fast Stop
   #"[OUTPUT] Drive Fast Stop Command" := #"[COMMAND] Axis Fast Stop" OR NOT "Safety Relais";
END_REGION

REGION Network 27: Error Executing
   #"[MESSAGE] Error Executing" := (#MoveToRest OR #Automatic_Negative OR #Manual_Negative OR #Manual_Positive OR #Automatic_Positive) AND NOT #"[INPUT] Drive Ready" AND NOT #"[INPUT] E-STOP Check";
END_REGION
END_FUNCTION

FUNCTION "EncoderFeedback" : Void   // FC16, FBD
TITLE = EncoderFeedback Block
VERSION : 0.1
// stored: AutoNumber true, IsIECCheckEnabled false, UDAEnableTagReadback false
   VAR_INPUT
      CounterTag : Int;   // Connect to the CounterTag IW102
      Position_Offset : Real;   // Fill in the tolerance, when the axis approves the position. Above or below the desired position
      Pulsfactor : Real;   // Number of pulses after 360 degree turn of the axis.
      Position_Correction : Real;   // Small Position Correction for the Axis
      ReferenceRun_Command : Bool;   // Command of starting the referencerun
      ReferenceSwitch : Bool;   // ReferenceSwitch Mounted on Axis
      ReferencePosition : Int;   // Position where the index puls of the reference switch enters.
   END_VAR
   VAR_OUTPUT
      Scaled_Position : Real;   // Scaled Position scaled with Pulsfactor
      Actual_Enc_Pos : Real;   // Actual Encoder Position
      AxisDB_Connection : Real;   // Connection with Axis DB connection
   END_VAR
   VAR_TEMP
      Corrected_Axis_Pos : Real;
      Unscaled_Position : Int;   // Unscaled Position of the Encoder
      Unsc2 : Int;   // Unsc 2 position
      Act_Enc_Pos_Int : DInt;
      Scaled_Position_Real : Real;
      PosDint : DInt;
      Unscaled_Position_Real : Real;
      InternalCounter : Int;
      CalDifCounter : Int;
      Pos_Storage : Int;
      Pos_Diffrence : Int;
      Add_Pos : Int;
      Sub_Pos : Int;
      LessThanZero : Bool;
      LTZ_out : Int;
      StoredOldPosition : Int;
   END_VAR
BEGIN

REGION Network 1: SPARE
END_REGION

NETWORK
TITLE = Call the Countermodule
      L     #CounterTag;  //Van tellerkaart TAG Gelinkt aan IW102
      L     "PositionManagement".Data.CntPlsPrev;  //Vorige scan
      -D;
      T     "PositionManagement".Data.CntPlsDiff;  //Verschil

      L     "PositionManagement".Data.CntPlsDiff;  // Verschil groter dan nul?
      L     0;
      >D;
      JCN   chkneg;

      L     "PositionManagement".Data.CntPlsDiff;  //Verschil optellen bij actuele pulswaarde
      L     "PositionManagement".Data.CntPlsAct;
      +D;
      T     "PositionManagement".Data.CntPlsAct;
      JU    end;  //rest overslaan.

chkneg:L     "PositionManagement".Data.CntPlsDiff;  // Verschil groter dan nul?
      L     0;
      <D;
      JCN   end;
      L     -1;  //verschil positief maken
      *D;
      T     "PositionManagement".Data.CntPlsDiff;  //verschil positief

      L     "PositionManagement".Data.CntPlsAct;  //Verschil optellen bij actuele pulswaarde
      +D;
      T     "PositionManagement".Data.CntPlsAct;

end:  NOP   0;

      L     #CounterTag;
      T     "PositionManagement".Data.CntPlsPrev;


REGION Network 3: Store Old Position
